(* IEC 61131-3 sources: traffic-lights/PLC_TrafficLights/Class/SdiasManager (part 4) *)

    if pAccessHandle then
      pAccessHandle^ := 0;
    end_if;

    Success := FALSE;
  end_if;

END_FUNCTION

FUNCTION VIRTUAL SdiasManager::AddBroadCastAccessesToList
  VAR
    i : USINT;
  END_VAR

  // Memory for Access data is already held by SDIAS Manager, No need for pHelpAccess

  // count the data for the varan payload frames
  // Access type is control broadcast 2 Byte, Read 0 Byte
  if SupportedFeatures.TimeBroadCastSupported then
    for i := 0 to SDIAS_NR_TIMEBROADCAST_DOS - 1 do
      ISOWriteDO.Length += sizeof(t_SDIAS_ControlByte) + sizeof(UINT);  // control byte + data length
      ISOReadDO.Length  += sizeof(t_SDIAS_StateByte);                   // state byte
    end_for;
  end_if;

END_FUNCTION

FUNCTION VIRTUAL SdiasManager::CheckTimeBroadCastSupported
	VAR_OUTPUT
		bTimeBroadCastSupported 	: BOOL;
	END_VAR
  VAR
    tempCmd             : CmdStruct;
    _result             : results;
    retval              : iprStates;
  END_VAR

  // Countercheck
  bTimeBroadCastSupported := TRUE;

  // Check if broadcast command is supported by OS
  if ConnectionType = SDIAS_CON_LOCAL_uC then

    // OS is only needed for local SDIAS
    if (pSDIAS^.udVersion < SDIAS_CILVERSION_BROADCAST) then
      bTimeBroadCastSupported := FALSE;
    end_if;

  end_if;

  // Check if broadcast command is supported SDIAS Manager
  if FeatureInfo.ProtocolVersion < SDIAS_PROTOCOLVERSION_BROADCAST then
    bTimeBroadCastSupported := FALSE;
  end_if;

  // Timestamp of HWControl must be valid
  tempCmd.uiCmd := CMD_GET_HW_TIMESTAMP;
  tempCmd.aPara[0]$t_GetHwTimestampCmd.udVersion    := 1;
  tempCmd.aPara[0]$t_GetHwTimestampCmd.udCoreSelect := 0;

  _result.aData[0]$t_GetHwTimestampResult.udVersion := 0; // Init return Value incase command is not implemented in HWControl

  retval := ToBusInterface.NewInst(#tempCmd, #_result);

  if retval <> READY then
    bTimeBroadCastSupported := FALSE;
  elsif _result.aData[0]$t_GetHwTimestampResult.udVersion < 1 then
    bTimeBroadCastSupported := FALSE;
  end_if;

END_FUNCTION

FUNCTION VIRTUAL SdiasManager::ReceiveSDOResponse
	VAR_INPUT
		Command 	: t_SDIAS_SDO_Cmd;
		Offset 	: HINT;
		Length 	: USINT;
		Result 	: iprStates;
		pResponseBuffer 	: ^USINT;
		ResponseLength 	: USINT;
	END_VAR
	VAR_OUTPUT
		ret_code 	: iprStates;
	END_VAR

  ret_code := READY;

  case Command of
    SDIAS_SDO_CMD_REBUILD_SDIAS:
      // if it succeeded, check if we have something to do
      if Result = READY then
        // everthing is fine
      else
        // an error occured while performing the operation
#ifdef HWC_LogError
        HWC_LogError(this, "@0083 (SdiasManager::ReceiveSDOResponse) Rebuild SDIAS SDO command failed!");
#endif
      end_if;
    SDIAS_SDO_CMD_SET_NEW_END:
      // if it succeeded, check if we have something to do
      if Result = READY then
        // everthing is fine
        bReceivedNewEndRsp := TRUE;
      else
        // an error occured while performing the operation
#ifdef HWC_LogError
        HWC_LogError(this, "@0084 (SdiasManager::ReceiveSDOResponse) Set new DOL end command failed!");
#endif
      end_if;

  else
    ret_code := ERROR;
#ifdef HWC_LogError
    HWC_LogError(this, "@0085 (SdiasManager::ReceiveSDOResponse) Invalid command in SDO response!");
#endif
  end_case;

END_FUNCTION

FUNCTION VIRTUAL SdiasManager::AddSDOReq
	VAR_INPUT
		pCmdSvr 	: ^SvrChCmd;
		Command 	: t_SDIAS_SDO_Cmd;
		Place 	: USINT;
		CmdLength 	: USINT;
		pReqBuf 	: ^USINT;
	END_VAR
	VAR_OUTPUT
		sd_retval 	: DINT;
	END_VAR

  // protect via mutex because this can be called from different task priorities
  OS_MT_WAIT(pv_Mutex);

  // if the buffer is full, or the next element in the buffer is already in use
  if (SDOHandling.pWrite^.Command <> SDIAS_SDO_CMD_INVALID) then
    sd_retval := SDIAS_MAILBOX_FULL;
    OS_MT_SIGNAL(pv_Mutex);
    return;
  end_if;

  // check the pointer first (if needed)
  if CmdLength then
    if pReqBuf then
      _memcpy(ptr1:=#SDOHandling.pWrite^.ReqBufData, ptr2:=pReqBuf, cntr:=CmdLength);
    else
      sd_retval := SDIAS_INVALID_PARAM_DATA_BUFFER;
      OS_MT_SIGNAL(pv_Mutex);
      return;
    end_if;
  end_if;

  SDOHandling.pWrite^.pCallBackSvr := pCmdSvr;
  SDOHandling.pWrite^.NMTCommand := 0;
  SDOHandling.pWrite^.SDIASPlace := Place;
  SDOHandling.pWrite^.CmdLength := CmdLength;

  case Command of
    SDIAS_SDO_CMD_MEM_READ,
    SDIAS_SDO_CMD_MEM_WRITE,
    SDIAS_SDO_CMD_CTRL_READ,
    SDIAS_SDO_CMD_CTRL_WRITE:
//    SDIAS_SDO_CMD_SPI_READ,
//    SDIAS_SDO_CMD_SPI_WRITE:
      // store offset and length for read and write accesses
      SDOHandling.pWrite^.RdWrHead := pReqBuf^$t_SDIAS_SDO_RdWr_Head;
    SDIAS_SDO_CMD_SPI_READ,
    SDIAS_SDO_CMD_SPI_WRITE:

      // store offset and length for read and write accesses
      SDOHandling.pWrite^.RdWrHead := pReqBuf^$t_SDIAS_SDO_RdWr_Head;

  end_case;

  // command is the last thing to store, because it indicates a complete entry
  SDOHandling.pWrite^.Command := Command;

  // we increment our used entries in the buffer (only for debugging)
  SDOHandling.EntriesUsed     += 1;

  // after we successfully added this SDO, set the write pointer to the next element
  if SDOHandling.pWrite = SDOHandling.pLastEntry then
    SDOHandling.pWrite := SDOHandling.pRingBufMemStart;
  else
    SDOHandling.pWrite += sizeof(t_SDORingBufEntry);
  end_if;

  sd_retval := SDIAS_OK;

  OS_MT_SIGNAL(pv_Mutex);

END_FUNCTION

FUNCTION VIRTUAL SdiasManager::CyclicSDOHandling
  VAR
  	i,j           : USINT;
    FoundIt       : BOOL;
		Offset 	      : HINT;
		Length 	      : USINT;
    pTempChannel  : ^t_SDOChannel;
    TempChannel   : t_SDOChannel;
    pRingBufEntry : ^t_SDORingBufEntry;
    FirstFound    : USINT;
    LastFound     : USINT;
    Channels2Add  : DINT;
    StartIndex    : USINT;
    EndIndex      : USINT;
    pCmdSvr       : ^SvrChCmd;
  	tempCmd       : CmdStruct;
    _result       : results;
    ReceiveBuffer : ARRAY [0..127] OF USINT;
    ReceiveLength : UDINT;
    sd_retval     : DINT;
    TempUDINT     : UDINT;
    OldChannelNo  : USINT;
  END_VAR

  // protect via mutex because this can be called from different task priorities
  OS_MT_WAIT(pv_Mutex);

  if ConnectionType = SDIAS_CON_VIA_VARAN_uC then

    // check sdo response first. if a channel is ready it can be used for the next request

    // GET SDO RESPONSE
    if (AsyReadUsage = _NotUsed) | (AsyReadUsage = _UsedBySDO) then

      // if the AsyRdDO is used for polling, we check if we got a response
      if AsyReadUsage = _UsedBySDO then
        StartIndex := ((ASYReadDO.Offset - SDOHandling.OffsetSDOResp) / sizeof(t_SDOChannel))$USINT;
        EndIndex := StartIndex + (ASYReadDO.Length / sizeof(t_SDOChannel))$USINT - 1;
        Offset := 0;
        for i := StartIndex to EndIndex do
          if SDOHandling.aChannelData[i].WaitForResponse then
            // check for the response (copy only header first)
            _memcpy(ptr1:=#TempChannel, ptr2:=ASYReadDO.pData$^t_SDOChannel + Offset, cntr:=sizeof(t_SDOChannel) - sizeof(t_SDOChannel.Data));
            pRingBufEntry := SDOHandling.aChannelData[i].pActElement;

            // if the header info is mirrored, the SDO is ready
            if ((TempChannel.MessageCounter AND SDIAS_MASK_MESSAGE_COUNTER) = pRingBufEntry^.MessageCounter) &
               (TempChannel.SDIASPlace = pRingBufEntry^.SDIASPlace) &
               (TempChannel.Command$t_SDIAS_SDO_Cmd = pRingBufEntry^.Command) then

              // we got our response
              SDOHandling.aChannelData[i].WaitForResponse := FALSE;
              SDOHandling.EntriesUsed -= 1;

              // check for error
              if (TempChannel.MessageCounter AND SDIAS_MASK_GLOBAL_ERROR_FLAG) then
                tempCmd.aPara[3] := ERROR;
                // copy error info
                _memcpy(ptr1:=#TempChannel.Data, ptr2:=ASYReadDO.pData + t_SDOChannel.Data + Offset, cntr:=TempChannel.LengthOfData);

                // show error info
                case TempChannel.Data$DINT of
                  SDIAS_SDO_ERROR_INVALID_MSG_CNT:
#ifdef HWC_LogValue1
                    HWC_LogValue1(this, "@0086 (SdiasManager::CyclicSDOHandling) SDO Error 0x{0}: Invalid message counter", TempChannel.Data$UDINT);
#endif

                  SDIAS_SDO_ERROR_MSG_CNT_NOT_SUCCESSIVE:
#ifdef HWC_LogValue1
                    HWC_LogValue1(this, "@0087 (SdiasManager::CyclicSDOHandling) SDO Error 0x{0}: Message counter not successive", TempChannel.Data$UDINT);
#endif

                  SDIAS_SDO_ERROR_INVALID_CMD:
#ifdef HWC_LogValue1
                    HWC_LogValue1(this, "@0088 (SdiasManager::CyclicSDOHandling) SDO Error 0x{0}: Invalid command", TempChannel.Data$UDINT);
#endif

                  SDIAS_SDO_ERROR_INVALID_SUBCMD:
#ifdef HWC_LogValue1
                    HWC_LogValue1(this, "@0089 (SdiasManager::CyclicSDOHandling) SDO Error 0x{0}: Invalid subcommand", TempChannel.Data$UDINT);
#endif

                  SDIAS_SDO_ERROR_INVALID_PLACE:
#ifdef HWC_LogValue1
                    HWC_LogValue1(this, "@008A (SdiasManager::CyclicSDOHandling) SDO Error 0x{0}: Invalid SDIAS Place", TempChannel.Data$UDINT);
#endif

                  SDIAS_SDO_ERROR_INVALID_CMD_LENGTH:
#ifdef HWC_LogValue1
                    HWC_LogValue1(this, "@008B (SdiasManager::CyclicSDOHandling) SDO Error 0x{0}: Invalid length of data bytes", TempChannel.Data$UDINT);
#endif

                  SDIAS_SDO_ERROR_INVALID_ACCESS_OFFSET:
#ifdef HWC_LogValue1
                    HWC_LogValue1(this, "@008C (SdiasManager::CyclicSDOHandling) SDO Error 0x{0}: Invalid offset for access", TempChannel.Data$UDINT);
#endif

                  SDIAS_SDO_ERROR_INVALID_ACCESS_LENGTH:
#ifdef HWC_LogValue1
                    HWC_LogValue1(this, "@008D (SdiasManager::CyclicSDOHandling) SDO Error 0x{0}: Invalid length for access", TempChannel.Data$UDINT);
#endif

                  SDIAS_SDO_ERROR_INTERNAL_TIMEOUT:
#ifdef HWC_LogValue1
                    HWC_LogValue1(this, "@008E (SdiasManager::CyclicSDOHandling) SDO Error 0x{0}: Internal timeout", TempChannel.Data$UDINT);
#endif

                  SDIAS_SDO_ERROR_GENERAL_ERROR:
#ifdef HWC_LogValue1
                    HWC_LogValue1(this, "@008F (SdiasManager::CyclicSDOHandling) SDO Error 0x{0}: General Error", TempChannel.Data$UDINT);
#endif

                  SDIAS_SDO_ERROR_MSG_CNT_CHANGED:
#ifdef HWC_LogValue1
                    HWC_LogValue1(this, "@0090 (SdiasManager::CyclicSDOHandling) SDO Error 0x{0}: Message counter changed while SDO request was processed", TempChannel.Data$UDINT);
#endif

                  SDIAS_SDO_ERROR_CLIENT_NOT_READY:
#ifdef HWC_LogValue1
                    HWC_LogValue1(this, "@0091 (SdiasManager::CyclicSDOHandling) SDO Error 0x{0}: Communication error between SDIAS Manager and SDIAS Client", TempChannel.Data$UDINT);
#endif

                  SDIAS_SDO_ERROR_MNG_DPRAM_FAILURE:
#ifdef HWC_LogValue1
                    HWC_LogValue1(this, "@0092 (SdiasManager::CyclicSDOHandling) SDO Error 0x{0}: Error accessing the SDIAS Manager DPRAM", TempChannel.Data$UDINT);
#endif

                  SDIAS_SDO_ERROR_ACCESS_NOT_ALLOWED:
#ifdef HWC_LogValue1
                    HWC_LogValue1(this, "@0093 (SdiasManager::CyclicSDOHandling) SDO Error 0x{0}: Access not allowed (e.g. control access to SDIAS Manager)", TempChannel.Data$UDINT);
#endif

                  SDIAS_SDO_ERROR_FLASH_ACCESS_FAILED:
#ifdef HWC_LogValue1
                    HWC_LogValue1(this, "@0094 (SdiasManager::CyclicSDOHandling) SDO Error 0x{0}: Flash access failed", TempChannel.Data$UDINT);
#endif

                  SDIAS_SDO_ERROR_INVALID_PARAMETERS:
#ifdef HWC_LogValue1
                    HWC_LogValue1(this, "@0095 (SdiasManager::CyclicSDOHandling) SDO Error 0x{0}: Invalid parameters in SDO request", TempChannel.Data$UDINT);
#endif

                else
#ifdef HWC_LogValue1
                  HWC_LogValue1(this, "@0096 (SdiasManager::CyclicSDOHandling) SDO Error 0x{0}: Unknown Error", TempChannel.Data$UDINT);
#endif
                end_case;
              else
                tempCmd.aPara[3]$iprStates := READY;
                // copy response data
                if TempChannel.LengthOfData then
                  if TempChannel.LengthOfData <= sizeof(t_SDOChannel.Data) then
                    _memcpy(ptr1:=#TempChannel.Data, ptr2:=ASYReadDO.pData + t_SDOChannel.Data + Offset, cntr:=TempChannel.LengthOfData);
                  else
#ifdef HWC_LogValue2
                    HWC_LogValue2(this, "@0097 (SdiasManager::CyclicSDOHandling) SDO Error: Length in response is too big (0x{0} Byte; Max: 0x{1} Byte)", TempChannel.LengthOfData, sizeof(t_SDOChannel.Data));
#endif
                  end_if;
                end_if;
              end_if;

              // if there is a response, distribute it and set this channel to "available for the next SDO" (set command to SDIAS_SDO_CMD_INVALID and pChannel to NIL)
              tempCmd.uiCmd := SDIAS_CMD_SDO_RESPONSE;
              tempCmd.aPara[0] := TempChannel.Command$t_SDIAS_SDO_Cmd;

              // if we got response data
              if TempChannel.LengthOfData then

                // if the SDO command was successful
                if tempCmd.aPara[3]$iprStates = READY then

                  // check if it's a command with offset and length info
                  case TempChannel.Command$t_SDIAS_SDO_Cmd of
                    SDIAS_SDO_CMD_MEM_READ,
                    SDIAS_SDO_CMD_MEM_WRITE,
                    SDIAS_SDO_CMD_CTRL_READ,
                    SDIAS_SDO_CMD_CTRL_WRITE:
                      // save header info in extra parameters
                      tempCmd.aPara[1] := pRingBufEntry^.RdWrHead.Offset;
                      tempCmd.aPara[2] := pRingBufEntry^.RdWrHead.Length;

                      // remove header info for user from payload
                      TempChannel.LengthOfData -= sizeof(t_SDIAS_SDO_RdWr_Head);

                      // pointer to data
                      tempCmd.aPara[4] := (#TempChannel.Data + sizeof(t_SDIAS_SDO_RdWr_Head))$DINT;

                    SDIAS_SDO_CMD_SPI_READ,
                    SDIAS_SDO_CMD_SPI_WRITE:

                      // no length or offset available
                      tempCmd.aPara[1] := 0;
                      tempCmd.aPara[2] := 0;

                      // pointer to data
                      tempCmd.aPara[4] := (#TempChannel.Data)$DINT;

                  else
                      // no length or offset available
                      tempCmd.aPara[1] := 0;
                      tempCmd.aPara[2] := 0;

                      // pointer to data
                      tempCmd.aPara[4] := (#TempChannel.Data)$DINT;
                  end_case;
                else
                  // check if it's a command with offset and length info
                  case TempChannel.Command$t_SDIAS_SDO_Cmd of
                    SDIAS_SDO_CMD_MEM_READ,
                    SDIAS_SDO_CMD_MEM_WRITE,
                    SDIAS_SDO_CMD_CTRL_READ,
                    SDIAS_SDO_CMD_CTRL_WRITE,
                    SDIAS_SDO_CMD_SPI_READ,
                    SDIAS_SDO_CMD_SPI_WRITE:
                      // save header info in extra parameters
                      tempCmd.aPara[1] := pRingBufEntry^.RdWrHead.Offset;
                      tempCmd.aPara[2] := pRingBufEntry^.RdWrHead.Length;
                  end_case;

                  // pointer to error code
                  tempCmd.aPara[4] := (#TempChannel.Data)$DINT;
                end_if;
              else
                tempCmd.aPara[4] := 0;
              end_if;
              tempCmd.aPara[5] := TempChannel.LengthOfData;

              pCmdSvr := pRingBufEntry^.pCallBackSvr;

              if pCmdSvr$pVirtualBase^.NewInst(#tempCmd, #_result) <> READY then
#ifdef HWC_LogValue1
                HWC_LogValue1(this, "@0099 (SdiasManager::CyclicSDOHandling) SDO Error: Error of module at place 0x{0} while receiving the SDO reponse (which was an ErrorCode)", i);
#endif
              end_if;

              // the position in the ringbuffer is free again
              pRingBufEntry^.BusyChannelNo := 0;
              pRingBufEntry^.Command := SDIAS_SDO_CMD_INVALID;

              // the SDO channel on the module is free again
              SDOHandling.aChannelData[i].pActElement := NIL;

            elsif (ops.tAbsolute - SDOHandling.aChannelData[i].RequestTime) >= SDIAS_SDO_TIMEOUT then
              // the SDO request timed out (should not happen)
#ifdef HWC_LogValue1
              HWC_LogValue1(this, "@0098 (SdiasManager::CyclicSDOHandling) SDO Error: Timeout while waiting for answer of the SDIAS Manager µC (Channel {0} of range 1-3)", i+1);
#endif

              // we got our response
              SDOHandling.aChannelData[i].WaitForResponse := FALSE;
              SDOHandling.EntriesUsed -= 1;

              // distribute timeout error and set this channel to "available for the next SDO" (set command to SDIAS_SDO_CMD_INVALID and pChannel to NIL)
              tempCmd.uiCmd := SDIAS_CMD_SDO_RESPONSE;
              tempCmd.aPara[0] := pRingBufEntry^.Command$UINT;

              // check if it's a command with offset and length info
              case pRingBufEntry^.Command of
                SDIAS_SDO_CMD_MEM_READ,
                SDIAS_SDO_CMD_MEM_WRITE,
                SDIAS_SDO_CMD_CTRL_READ,
                SDIAS_SDO_CMD_CTRL_WRITE,
                SDIAS_SDO_CMD_SPI_READ,
                SDIAS_SDO_CMD_SPI_WRITE:
                  // save header info in extra parameters
                  tempCmd.aPara[1] := pRingBufEntry^.RdWrHead.Offset;
                  tempCmd.aPara[2] := pRingBufEntry^.RdWrHead.Length;
              else
                  // no length or offset available
                  tempCmd.aPara[1] := 0;
                  tempCmd.aPara[2] := 0;
              end_case;

              tempCmd.aPara[3] := ERROR;
              tempCmd.aPara[4] := 0;
              tempCmd.aPara[5] := 0; // no data available

              pCmdSvr := pRingBufEntry^.pCallBackSvr;
              if pCmdSvr$pVirtualBase^.NewInst(#tempCmd, #_result) <> READY then
#ifdef HWC_LogValue1
                HWC_LogValue1(this, "@0099 (SdiasManager::CyclicSDOHandling) SDO Error: Error of module at place 0x{0} while receiving the SDO reponse", i);
#endif
              end_if;

              // the position in the ringbuffer is free again
              pRingBufEntry^.BusyChannelNo := 0;
              pRingBufEntry^.Command := SDIAS_SDO_CMD_INVALID;

              // the SDO channel on the module is free again
              SDOHandling.aChannelData[i].pActElement := NIL;
            end_if;
          end_if;

          Offset += sizeof(t_SDOChannel);
        end_for;
      end_if;

      // check for the first (needed for offset) and last (needed for length)
      Length := 0;
      FoundIt := FALSE;
      for i := 0 to (SDIAS_SDO_CHANNEL_NO-1) do
        if SDOHandling.aChannelData[i].pActElement & SDOHandling.aChannelData[i].WaitForResponse then
          if FoundIt = FALSE then
            // found first used channel
            FoundIt := TRUE;
            Offset := SDOHandling.OffsetSDOResp + i * sizeof(t_SDOChannel);
          end_if;
          Length += sizeof(t_SDOChannel);
        end_if;
      end_for;

      if FoundIt then

        // if we have pending SDO requests, start the AsyRdDO for polling
        if ChangeAsyRd(Offset:=Offset,
                       Length:=Length,
                       RunState:=_BUS_IF_RUN_STATE_CONT_RUN,
                       UsageType:=_UsedBySDO) = FALSE then
#ifdef HWC_LogError
          HWC_LogError(this, "@009A (SdiasManager::CyclicSDOHandling) Error occured at starting the ReadDO for SDO polling");
#endif
        end_if;
      else
        // if all pending SDOs received stop DO
        if AsyReadUsage = _UsedBySDO then
          if ChangeAsyRd(Offset:=0,
                         Length:=0,
                         RunState:=_BUS_IF_RUN_STATE_NO_RUN,
                         UsageType:=_UsedBySDO) = FALSE then
#ifdef HWC_LogError
          HWC_LogError(this, "@009B (SdiasManager::CyclicSDOHandling) Error occured at stopping the ReadDO");
#endif
          end_if;
        end_if;
      end_if;
    end_if;

    // SEND SDO REQUEST
    if (AsyWriteUsage = _NotUsed) | (AsyWriteUsage = _UsedBySDO) then
      // if there is a free channel on the module, we have unsent requests and the AsyWrDO is not used => send the Request (or more than 1 if possible)

      // first check if we need to increment the msg counter for a previously sent SDO message
      if SDOHandling.IncrementMsgCnt then
        for i := 0 to (SDIAS_SDO_CHANNEL_NO-1) do
          if SDOHandling.IncrementMsgCnt AND 1 then
            // next message counter for this channel
            if SDOHandling.aChannelData[i].MessageCnt = SDIAS_MASK_MESSAGE_COUNTER then
              SDOHandling.aChannelData[i].MessageCnt    := 0;
            else
              SDOHandling.aChannelData[i].MessageCnt    += 1;
            end_if;

            SDOHandling.aChannelData[i].pActElement^.MessageCounter := SDOHandling.aChannelData[i].MessageCnt;
            pTempChannel := #SDOHandling.aChannelData[i].ChannelData;
            pTempChannel^.MessageCounter  := SDOHandling.aChannelData[i].MessageCnt;

            // save the new message counter to the Varan DO
            _memcpy(ptr1:=ASYWriteDO.pData$^USINT + i * sizeof(t_SDOChannel) - (ASYWriteDO.Offset - SDOHandling.OffsetSDOReq)$USINT, ptr2:=pTempChannel, cntr:=pTempChannel^.LengthOfData + sizeof(t_SDOChannel) - sizeof(t_SDOChannel.Data));
            SDOHandling.aChannelData[i].WaitForResponse := TRUE;
            TempUDINT := ops.tAbsolute;
            SDOHandling.aChannelData[i].RequestTime     := TempUDINT;
          end_if;
          SDOHandling.IncrementMsgCnt := SDOHandling.IncrementMsgCnt SHR 1;
        end_for;

        // use the same length and offset (it's the same frame just with different message counters)
        Offset := ASYWriteDO.Offset;
        Length := ASYWriteDO.Length$USINT;

        // write the same frame again with higher message counter on the modified SDOs
        if ChangeAsyWr(Offset:=Offset,
                       Length:=Length,
                       RunState:=_BUS_IF_RUN_STATE_CONT_RUN,
                       UsageType:=_UsedBySDO) = FALSE then
#ifdef HWC_LogError
          HWC_LogError(this, "@009C (SdiasManager::CyclicSDOHandling) Error occured at starting the WriteDO to write the new message counter");
#endif
        end_if;
      else
        // check for a free channel
        FoundIt := FALSE;
        for i := 0 to (SDIAS_SDO_CHANNEL_NO-1) do
          if SDOHandling.aChannelData[i].pActElement = NIL then
            // found a free channel
            FoundIt := TRUE;
            FirstFound := LastFound := i;
            Offset := SDOHandling.OffsetSDOReq + i * sizeof(t_SDOChannel);
            exit;
          end_if;
        end_for;

        // now we fill the buffer in the channels of the hardware (continue as long as there is space in the buffer and we have SDOs to send)
        Channels2Add := 0;
        while FoundIt & (SDOHandling.pRead^.Command <> SDIAS_SDO_CMD_INVALID) & (SDOHandling.pRead^.BusyChannelNo = 0) do
          // i is the index of the free channel => add the data
          pTempChannel := #SDOHandling.aChannelData[i].ChannelData;
          SDOHandling.aChannelData[i].pActElement     := SDOHandling.pRead;
          SDOHandling.pRead^.MessageCounter           := SDOHandling.aChannelData[i].MessageCnt;
          pTempChannel^.MessageCounter                := SDOHandling.pRead^.MessageCounter;
          pTempChannel^.NMT                           := SDOHandling.pRead^.NMTCommand;
          pTempChannel^.SDIASPlace                    := SDOHandling.pRead^.SDIASPlace;
          pTempChannel^.Command$t_SDIAS_SDO_Cmd       := SDOHandling.pRead^.Command;
          pTempChannel^.LengthOfData                  := SDOHandling.pRead^.CmdLength;
          if pTempChannel^.LengthOfData then
            _memcpy(ptr1:=#pTempChannel^.Data, ptr2:=#SDOHandling.pRead^.ReqBufData, cntr:=pTempChannel^.LengthOfData);
          end_if;

          // put the SDO request into the DPRAM on the right channel
          _memcpy(ptr1:=ASYWriteDO.pData$^t_SDOChannel + Channels2Add * sizeof(t_SDOChannel), ptr2:=pTempChannel, cntr:=pTempChannel^.LengthOfData + sizeof(t_SDOChannel) - sizeof(t_SDOChannel.Data));

          // remember this as the last found SDO to work with
          LastFound := i;

          // remember that we have to increment the message counter here
          SDOHandling.IncrementMsgCnt := SDOHandling.IncrementMsgCnt OR (1 SHL i);

          // this element is done by channel x
          SDOHandling.pRead^.BusyChannelNo := i+1;

          // increase channels to add
          Channels2Add += 1;

          // after we successfully added this SDO, set the read pointer to the next element
          if SDOHandling.pRead = SDOHandling.pLastEntry then
            SDOHandling.pRead := SDOHandling.pRingBufMemStart;
          else
            SDOHandling.pRead += sizeof(t_SDORingBufEntry);
          end_if;

          OldChannelNo := i;

          // check for a free channel
          FoundIt := FALSE;
          for i := 0 to (SDIAS_SDO_CHANNEL_NO-1) do
            if SDOHandling.aChannelData[i].pActElement = NIL then
              // found a free channel
              FoundIt := TRUE;

              if i > (OldChannelNo + 1) then
                // refresh the data in the DPRAM for the skipped channels
                for j := (OldChannelNo+1) to (i-1) do
                  // put the SDO request into the DPRAM on the right channel
                  _memcpy(ptr1:=ASYWriteDO.pData$^t_SDOChannel + j * sizeof(t_SDOChannel), ptr2:=#SDOHandling.aChannelData[j].ChannelData, cntr:=SDOHandling.aChannelData[j].ChannelData.LengthOfData + sizeof(t_SDOChannel) - sizeof(t_SDOChannel.Data));

                  // increase channels to add, because we also write the skipped ones
                  Channels2Add += 1;
                end_for;
              end_if;

              exit;
            end_if;
          end_for;
        end_while;

        if Channels2Add then
          Length := (LastFound - FirstFound + 1)$USINT * sizeof(t_SDOChannel);
          // if we have something to write => write it
          if ChangeAsyWr(Offset:=Offset,
                         Length:=Length,
                         RunState:=_BUS_IF_RUN_STATE_CONT_RUN,
                         UsageType:=_UsedBySDO) = FALSE then
#ifdef HWC_LogError
            HWC_LogError(this, "@009D (SdiasManager::CyclicSDOHandling) Error occured at starting the WriteDO to write the new SDO command");
#endif
          end_if;
        elsif AsyWriteUsage = _UsedBySDO then
          // otherwise release the write buffer to other purposes
          if ChangeAsyWr(Offset:=0,
                         Length:=0,
                         RunState:=_BUS_IF_RUN_STATE_NO_RUN,
                         UsageType:=_UsedBySDO) = FALSE then
#ifdef HWC_LogError
            HWC_LogError(this, "@009E (SdiasManager::CyclicSDOHandling) Error occured at stopping the WriteDO");
#endif
          end_if;
        end_if;
      end_if;
    end_if;
  else
    // if connected locally we can use the OS interfaces to access the SDO channels

    // check sdo response first. if a channel is ready it can be used for the next request

    // GET SDO RESPONSE
    if SDOHandling.EntriesUsed then
      // post init blocks the tasks in cyclic priority (the SDIAS Manager Code is running in lower priority than cyclic and has no time during the postinit) => give it some time
      if (b_PostInitFinished = FALSE) then
        ToMultiTask.TASKDELAY(timeout0:=SDIAS_WAIT_TIME_IN_POST_INIT);
      end_if;
      // check if we got a response
      for i := 0 to (SDIAS_SDO_CHANNEL_NO-1) do
        if SDOHandling.aChannelData[i].WaitForResponse then

          // get the SDO response
          ReceiveLength := 0;
          sd_retval := SDIAS_iReadSdoResponseChannel(udSdoHandle       := SDOHandling.aChannelData[i].SdoHandle
                                                   , udBufferLength    := sizeof(ReceiveBuffer)
                                                   , pucData           := #ReceiveBuffer[0]
                                                   , pudDataLength     := #ReceiveLength
                                                   );

          // check if it's finished => no more busy
          if sd_retval <> SDIAS_SDO_REQUEST_BUSY then
            if ReceiveLength <= sizeof(TempChannel.Data) then
              pRingBufEntry := SDOHandling.aChannelData[i].pActElement;

              // copy the info
              _memcpy(ptr1:= #TempChannel.Data, ptr2:= #ReceiveBuffer[0], cntr:= ReceiveLength);
              TempChannel.LengthOfData := ReceiveLength$USINT;
              TempChannel.Command$t_SDIAS_SDO_Cmd := pRingBufEntry^.Command;

              // we got our response
              SDOHandling.aChannelData[i].WaitForResponse := FALSE;
              SDOHandling.EntriesUsed -= 1;

              // check for error
              if sd_retval <> SDIAS_OK then
                tempCmd.aPara[3] := ERROR;

                LogSDOErrorInfo(sd_retval);
              else
                tempCmd.aPara[3]$iprStates := READY;
              end_if;

              // if there is a response, distribute it and set this channel to "available for the next SDO" (set command to SDIAS_SDO_CMD_INVALID and pChannel to NIL)
              tempCmd.uiCmd := SDIAS_CMD_SDO_RESPONSE;
              tempCmd.aPara[0] := pRingBufEntry^.Command$INT;

              // if we got response data
              if TempChannel.LengthOfData then

                // if the SDO command was successful
                if tempCmd.aPara[3]$iprStates = READY then

                  // check if it's a command with offset and length info
                  case TempChannel.Command$t_SDIAS_SDO_Cmd of
                    SDIAS_SDO_CMD_MEM_READ,
                    SDIAS_SDO_CMD_MEM_WRITE,
                    SDIAS_SDO_CMD_CTRL_READ,
                    SDIAS_SDO_CMD_CTRL_WRITE:
                      // save header info in extra parameters
                      tempCmd.aPara[1] := pRingBufEntry^.RdWrHead.Offset;
                      tempCmd.aPara[2] := pRingBufEntry^.RdWrHead.Length;

                      // remove header info for user from payload
                      TempChannel.LengthOfData -= sizeof(t_SDIAS_SDO_RdWr_Head);

                      // pointer to data
                      tempCmd.aPara[4] := (#TempChannel.Data + sizeof(t_SDIAS_SDO_RdWr_Head))$DINT;

                    SDIAS_SDO_CMD_SPI_READ,
                    SDIAS_SDO_CMD_SPI_WRITE:
                      // no length or offset available
                      tempCmd.aPara[1] := 0;
                      tempCmd.aPara[2] := 0;

                      // pointer to data
                      tempCmd.aPara[4] := (#TempChannel.Data)$DINT;

                  else
                      // no length or offset available
                      tempCmd.aPara[1] := 0;
                      tempCmd.aPara[2] := 0;

                      // pointer to data
                      tempCmd.aPara[4] := (#TempChannel.Data)$DINT;
                  end_case;
                else
                  // check if it's a command with offset and length info
                  case TempChannel.Command$t_SDIAS_SDO_Cmd of
                    SDIAS_SDO_CMD_MEM_READ,
                    SDIAS_SDO_CMD_MEM_WRITE,
                    SDIAS_SDO_CMD_CTRL_READ,
                    SDIAS_SDO_CMD_CTRL_WRITE,
                    SDIAS_SDO_CMD_SPI_READ,
                    SDIAS_SDO_CMD_SPI_WRITE:
                      // save header info in extra parameters
                      tempCmd.aPara[1] := pRingBufEntry^.RdWrHead.Offset;
                      tempCmd.aPara[2] := pRingBufEntry^.RdWrHead.Length;
                  end_case;

                  // pointer to error code
                  tempCmd.aPara[4] := (#sd_retval)$DINT;
                end_if;
              else
                tempCmd.aPara[4] := 0;
              end_if;
              tempCmd.aPara[5] := TempChannel.LengthOfData;

              pCmdSvr := pRingBufEntry^.pCallBackSvr;
              if pCmdSvr$pVirtualBase^.NewInst(#tempCmd, #_result) <> READY then
#ifdef HWC_LogValue1
                HWC_LogValue1(this, "@0099 (SdiasManager::CyclicSDOHandling) SDO Error: Error of module at place 0x{0} while receiving the SDO reponse (which was an ErrorCode)", i);
#endif
              end_if;

              // the position in the ringbuffer is free again
              pRingBufEntry^.BusyChannelNo := 0;
              pRingBufEntry^.Command := SDIAS_SDO_CMD_INVALID;

              // the SDO channel on the module is free again
              SDOHandling.aChannelData[i].pActElement := NIL;
            else
#ifdef HWC_LogValue2
              HWC_LogValue2(this, "@009F (SdiasManager::CyclicSDOHandling) SDO Response too big. Received 0x{0} bytes. Maximum is 0x{1} bytes.", ReceiveLength, sizeof(TempChannel.Data));
#endif
            end_if;
          end_if;
        end_if;
      end_for;
    end_if;

    // SEND SDO REQUEST
    if SDOHandling.EntriesUsed then
      // if there is a free channel on the module and we have unsent requests => send the Requests

      // check for a free channel
      FoundIt := FALSE;
      for i := 0 to (SDIAS_SDO_CHANNEL_NO-1) do
        if SDOHandling.aChannelData[i].pActElement = NIL then
          // found a free channel
          FoundIt := TRUE;
          FirstFound := LastFound := i;
          exit;
        end_if;
      end_for;

      // now we fill the buffer in the channels of the hardware (continue as long as there is space in the buffer and we have SDOs to send)
      while FoundIt & (SDOHandling.pRead^.Command <> SDIAS_SDO_CMD_INVALID) & (SDOHandling.pRead^.BusyChannelNo = 0) do
        // i is the index of the free channel => add the data
        SDOHandling.aChannelData[i].pActElement     := SDOHandling.pRead;
        SDOHandling.pRead^.MessageCounter           := SDOHandling.aChannelData[i].MessageCnt;
        TempChannel.MessageCounter                  := SDOHandling.pRead^.MessageCounter;
        TempChannel.NMT                             := SDOHandling.pRead^.NMTCommand;
        TempChannel.SDIASPlace                      := SDOHandling.pRead^.SDIASPlace;
        TempChannel.Command$t_SDIAS_SDO_Cmd         := SDOHandling.pRead^.Command;
        TempChannel.LengthOfData                    := SDOHandling.pRead^.CmdLength;
        if TempChannel.LengthOfData then
          _memcpy(ptr1:=#TempChannel.Data, ptr2:=#SDOHandling.pRead^.ReqBufData, cntr:=TempChannel.LengthOfData);
        end_if;

        // send the SDO to the OS Interface
        sd_retval := SDIAS_iSendSdoRequestChannel(hManagerNodeHandle:= udNodeHandle
                                                , udChannel         := i
                                                , udCommand         := TempChannel.Command$t_SDIAS_SDO_Cmd
                                                , udSdiasAddress    := TempChannel.SDIASPlace
                                                , udDataLength      := TempChannel.LengthOfData
                                                , pucData           := #TempChannel.Data[0]
                                                , pudSdoHandle      := #SDOHandling.aChannelData[i].SdoHandle
                                                );

        if sd_retval = SDIAS_OK then
          // this element is done by channel x
          SDOHandling.pRead^.BusyChannelNo := i+1;

          SDOHandling.aChannelData[i].WaitForResponse := TRUE;
          TempUDINT := ops.tAbsolute;
          SDOHandling.aChannelData[i].RequestTime     := TempUDINT;

          // after we successfully added this SDO, set the read pointer to the next element
          if SDOHandling.pRead = SDOHandling.pLastEntry then
            SDOHandling.pRead := SDOHandling.pRingBufMemStart;
          else
            SDOHandling.pRead += sizeof(t_SDORingBufEntry);
          end_if;

          // check for a free channel
          FoundIt := FALSE;
          for i := 0 to (SDIAS_SDO_CHANNEL_NO-1) do
            if SDOHandling.aChannelData[i].pActElement = NIL then
              // found a free channel
              FoundIt := TRUE;
              exit;
            end_if;
          end_for;
        else
          LogSDOErrorInfo(sd_retval);
          exit;
        end_if;
      end_while;
    end_if;
  end_if;

    OS_MT_SIGNAL(pv_Mutex);

END_FUNCTION

FUNCTION VIRTUAL SdiasManager::SetRequiredError
	VAR_INPUT
		pTargetThis 	: ^SdiasBase;(* := NIL *)
		Place 	: UDINT;(* := SDIAS_PLACE_NO_MODULE_ADDED_SO_FAR *)
	END_VAR
  VAR
  	tempCmd         : CmdStruct;
    _result         : results;
    i : UDINT;
    FoundIt : BOOL;
  END_VAR

  if pTargetThis & (Place <> SDIAS_PLACE_NO_MODULE_ADDED_SO_FAR) then
    pTargetThis^.ClassState := _RequiredError;

#ifdef HWC_LogValue1
    HWC_LogValue1(this, "@00A0 (SdiasManager::SetRequiredError) Required Error on SDIAS Place 0x{0}", Place);
#endif
  else
    // general required error (initialisation failed) => search for the first required module to blame (if there is one)
    FoundIt := FALSE;
    if MaxPlace <> SDIAS_PLACE_NO_MODULE_ADDED_SO_FAR then
      for i := 0 to MaxPlace do
        if ModuleObjInfo[i].pThis & ModuleObjInfo[i].Required then
          FoundIt := TRUE;
        end_if;
      end_for;
    end_if;

    // if no required module => don't crash
    if FoundIt = FALSE then
      return;
    end_if;
  end_if;

  ClassState := _RequiredError;

  // set required error
  tempCmd.uiCmd     := _BUS_IF_SET_REQUIRED_ERROR;

  ToBusInterface.NewInst(pPara:=#tempCmd, pResult:=#_result);
  if _result.aData[0]$t_BusIFRetvalErrorcode <> _BUS_IF_RETVAL_OK then
#ifdef HWC_LogError
    HWC_LogError(this, "@00A1 (SdiasManager::SetRequiredError) Failed to set required error to BusInterface");
#endif
  end_if;

  if InitSSW <> _PrepareError then
    ErrorInitStep := InitSSW;
    InitSSW := _PrepareError;
  end_if;

END_FUNCTION

// New interface - 2013-05-28
// -----------------------------------------------------------------------
// -	bIsWriteAcc0 : 0 - read access , 1 - write access
// -	iModAddr0 : Module adress at sdias bus (device adr + offset)
// -	iDataLen0 : Data length
// -	bCtrlAcc0 : 0 - access to regular memory, 1 > access to ctrl access
// -    bAccList0 : 0 - access to iso read/write list, 1 - acc to manager admin list, 2 - access to sdo list, 3 - access to periodic manager list

FUNCTION VIRTUAL SdiasManager::DOL_Handling_Add_DO_TO_List
	VAR_INPUT
		bIsWriteAcc0 	: BOOL;
		usModulePlace0 	: USINT;
		iModAddr0 	: HINT;
		iDataLen0 	: UINT;
		bCtrlAcc0 	: BOOL;
		iWaitDOOffset0 	: UINT;
		bIsDynamic0 	: BOOL;
		pActAccess0 	: ^t_AccessElement;
		bIsBroadCast 	: BOOL;(* := FALSE *)
	END_VAR
	VAR_OUTPUT
		iRetCode 	: DINT;
	END_VAR
  VAR
    pReadList       : ^t_SDIAS_DOL_DESC;
    pWriteList      : ^t_SDIAS_DOL_DESC;
    iEndDataPointRd : UINT;
    iEndDOLPointRd  : UDINT;
    iEndDataPointWr : UINT;
    iEndDOLPointWr  : UDINT;
    udCmdType       : UDINT;
    ReadLen         : UINT;
    ReadAdd         : HDINT;
    WriteLen        : UINT;
    WriteAdd        : HDINT;
    udDOFlags       : UDINT;
    bIsFarAccess    : BOOL;
    usBlockNo1k     : USINT;
    usRetries       : BSINT;
    dolType         : UDINT;
  END_VAR

  iRetCode := -1;

  (* Only ISO DOL	in hardware classes *)
  pReadList := #gcRead_DOL_Desc;
  pWriteList := #gcWrite_DOL_Desc;

  // calculate the module address for far accesses and other
  if pActAccess0^.bIsFarAcc then
    bIsFarAccess  := TRUE;
    usBlockNo1k   := to_usint(iModAddr0 shr 10);
    iModAddr0     := (iModAddr0 AND 16#3FF) + (usModulePlace0 shl 10);
  else
    bIsFarAccess  := FALSE;
    usBlockNo1k   := 0;
    iModAddr0     := iModAddr0 + (usModulePlace0 shl 10);
  end_if;

  if ConnectionType = SDIAS_CON_VIA_VARAN_uC then

    (*	Check endpoints of data and DOL	*)
    iEndDataPointRd := pReadList^.iBaseAddrData + pReadList^.iOffLastData + 1;
    iEndDOLPointRd  := pReadList^.iBaseAddr + pReadList^.iOffEndCmd;

    iEndDataPointWr := pWriteList^.iBaseAddrData + pWriteList^.iOffLastData +  1;
    iEndDOLPointWr  := pWriteList^.iBaseAddr + pWriteList^.iOffEndCmd;

    if(bIsWriteAcc0 = 0) then
      (*	Check endpoints of data and DOL	*)
      iEndDataPointRd += iDataLen0;
      iEndDOLPointRd  += sizeof(t_SDIAS_STD_CMD_DO);
    else
      (*	Check endpoints of data and DOL	*)
      iEndDataPointWr += iDataLen0;
      iEndDOLPointWr  += sizeof(t_SDIAS_STD_CMD_DO);
    end_if;

    (* Check available data	in read space *)
    if(iEndDataPointRd > pReadList^.iEndAddrData) then
      iRetCode := -3;
    (* Check space in DOL	*)
    elsif(iEndDOLPointRd > pReadList^.iEndAddr) then
      iRetCode := -4;
    (* Check available data	in write space *)
    elsif(iEndDataPointWr > pWriteList^.iEndAddrData) then
      iRetCode := -5;
    (* Check space in DOL	*)
    elsif(iEndDOLPointWr > pWriteList^.iEndAddr) then
      iRetCode := -6;
    (* Space for all required data	*)
    else

      // Add 1 to switch to first empty byte
      pWriteList^.iOffLastData += sizeof(t_SDIAS_ControlByte);										(* Add do ctrl byte to data		*)
      pReadList^.iOffLastData += sizeof(t_SDIAS_StateByte);

      pWriteList^.iOffFirstData := pWriteList^.iOffLastData;			(* Store data start points		*)
      pReadList^.iOffFirstData := pReadList^.iOffLastData;

      // dynamic accesses need more bytes in the write payload
      if bIsDynamic0 then
        // control byte is already considered, so we have to add the difference here
        pWriteList^.iOffLastData += (sizeof(t_SDIAS_ControlStructDynamic) - sizeof(t_SDIAS_ControlByte));
      end_if;

      cModulAccessCmds[0].OffsetWritePayload := pWriteList^.iBaseAddrData + pWriteList^.iOffFirstData;		(* Store data offsets			*)
      cModulAccessCmds[0].OffsetReadPayload := pReadList^.iBaseAddrData + pReadList^.iOffFirstData;

      (* Set wait for DO to inactive	*)
      cModulAccessCmds[0].OffsetVolatileWaitFlag := iWaitDOOffset0;

      (* Init scratchpad info to 0	*)
      cModulAccessCmds[0].ErrorInfo := 0;

      usRetries := SDIAS_RETRIES_ALLOWED;
      // No retries with Broadcast
      if bIsBroadCast then
        usRetries := 0;
      end_if;

      (* Ctrl access *)
      if(bCtrlAcc0 <> 0) then
        (* Ctrl access +  retrys	*)
        cModulAccessCmds[0].CmdRetries  := SDIAS_CMD_ACC_CONTROL + (usRetries shl 5);
      elsif bIsFarAccess then
        (* Mem far access +  retrys	*)
        cModulAccessCmds[0].CmdRetries  := SDIAS_CMD_ACC_MEMORY_FAR + (usRetries shl 5);
      else
        (* Mem access +  retrys	*)
        cModulAccessCmds[0].CmdRetries  := SDIAS_CMD_ACC_MEMORY + (usRetries shl 5);
      end_if;

      (* Init reserved info to 0	*)
      cModulAccessCmds[0].Reserved := 0;

      (* Write command to dpram 	*)
      if(bIsWriteAcc0 = 0) then
        if bIsFarAccess then
          cModulAccessCmds[0].ReadLength  := to_usint(iDataLen0);
          cModulAccessCmds[0].ReadOffset  := to_uint(iModAddr0);

          cModulAccessCmds[0].WriteLength := 0;
          cModulAccessCmds[0].WriteOffset := usBlockNo1k;
        else
          cModulAccessCmds[0].ReadLength := to_usint(iDataLen0);
          cModulAccessCmds[0].ReadOffset := to_uint(iModAddr0);

          cModulAccessCmds[0].WriteLength := 0;
          cModulAccessCmds[0].WriteOffset  := 0;
        end_if;

        (* Store write adress of new command  *)
        uiWriteCmdAddr := pReadList^.iBaseAddr + pReadList^.iOffEndCmd;

        (* Increment offset of end command	*)
        pReadList^.iOffEndCmd += sizeof(t_SDIAS_STD_CMD_DO);

        (* End of list	*)
        DOL_Handling_Create_End_Cmd(#cModulAccessCmds[1]);

        (* Add read length to iso read usage	*)
        pReadList^.iOffLastData += iDataLen0;

        (* Set usage vars	*)
        pReadList^.iUsageData := pReadList^.iOffLastData + 1;
        pReadList^.iUsageDOL := pReadList^.iOffEndCmd + sizeof(t_SDIAS_STD_CMD_DO);

        pWriteList^.iUsageData := pWriteList^.iOffLastData + 1;

      else
        if bIsFarAccess then
          cModulAccessCmds[0].ReadLength := 0;
          cModulAccessCmds[0].ReadOffset := usBlockNo1k;

          cModulAccessCmds[0].WriteLength := to_usint(iDataLen0);
          cModulAccessCmds[0].WriteOffset  := to_uint(iModAddr0);
        elsif bIsBroadCast then
          cModulAccessCmds[0]$t_SDIAS_BROADCAST_CMD_DO.iNoOfReadBytes   := 0;
          cModulAccessCmds[0]$t_SDIAS_BROADCAST_CMD_DO.iModAddrRdWrCmd  := to_uint(iModAddr0);
          cModulAccessCmds[0]$t_SDIAS_BROADCAST_CMD_DO.iCmdSubtype      := SDIAS_TIMEBROADCAST_SUBCMD;
          cModulAccessCmds[0]$t_SDIAS_BROADCAST_CMD_DO.iNoOfWriteBytes  := to_usint(iDataLen0);
        else
          cModulAccessCmds[0].ReadLength := 0;
          cModulAccessCmds[0].ReadOffset := 0;

          cModulAccessCmds[0].WriteLength := to_usint(iDataLen0);
          cModulAccessCmds[0].WriteOffset  := to_uint(iModAddr0);
        end_if;

        (* Store write adress of new command  *)
        uiWriteCmdAddr := pWriteList^.iBaseAddr + pWriteList^.iOffEndCmd;

        (* Increment offset of end command	*)
        pWriteList^.iOffEndCmd += sizeof(t_SDIAS_STD_CMD_DO);

        (* End of list	*)
        DOL_Handling_Create_End_Cmd(#cModulAccessCmds[1]);

        (* Add write length to iso write usage	*)
        pWriteList^.iOffLastData += iDataLen0;

        (* Set usage vars	*)
        pReadList^.iUsageData := pReadList^.iOffLastData + 1;

        pWriteList^.iUsageData := pWriteList^.iOffLastData + 1;
        pWriteList^.iUsageDOL := pWriteList^.iOffEndCmd + sizeof(t_SDIAS_STD_CMD_DO);

        (* Reset write payload	*)
        //SDIAS_Module_CPLD_Com_Write_Data(pWriteList^.iBaseAddrData + pWriteList^.iOffFirstData + 1, iDataLen0 , (void *)&iDOL_ResetData[0]);

      end_if;

      iRetCode := 0;

    end_if;

  else
    // locally we use the OS interface to create the DO

    (* Ctrl access *)
    if(bCtrlAcc0 <> 0) then
      (* Ctrl access +  retrys	*)
      udCmdType         := SDIAS_CMD_ACC_CONTROL;
    elsif  bIsFarAccess then
      // far memory access
      udCmdType         := SDIAS_CMD_ACC_MEMORY_FAR;
    else
      (* Mem access +  retrys	*)
      udCmdType         := SDIAS_CMD_ACC_MEMORY;
    end_if;

    // if the interface for dynamic DOs is not available => use the old interface
    if (pSDIAS^.udVersion < SDIAS_CIL_VERSION_SUPPORTS_DYNAMIC_DO) then
      iRetCode := SDIAS_iAddDo(hNodeHandle         := udNodeHandle
                             , udDolType           := SDIAS_DOL_TYPE_ISO
                             , udCmdType           := udCmdType
                             , udRetries           := SDIAS_RETRIES_ALLOWED
                             , udIsWriteAcc        := bIsWriteAcc0
                             , udModuleAddress     := iModAddr0
                             , udDataLen           := iDataLen0
                             , hAddrVolatileWait   := iWaitDOOffset0
                             , phAddrWriteData     := (#cModulAccessCmds[0].OffsetWritePayload)$^pVoid
                             , phAddrReadData      := (#cModulAccessCmds[0].OffsetReadPayload)$^pVoid
                             );

    else

        // make read and write settings
      if bIsWriteAcc0 then
        WriteLen := iDataLen0;
        WriteAdd := iModAddr0;
        ReadLen  := 0;
        ReadAdd  := usBlockNo1k;

        if bIsBroadCast then
          ReadAdd := iModAddr0; // RdWr Access with rd length 0
        end_if;

      else
        WriteLen := 0;
        WriteAdd := usBlockNo1k;
        ReadLen  := iDataLen0;
        ReadAdd  := iModAddr0;
      end_if;

      dolType   := SDIAS_DOL_TYPE_ISO;
      usRetries := SDIAS_RETRIES_ALLOWED;
      // set DO flags
      udDOFlags := 0;
      if bIsDynamic0 then
        if bIsFarAccess then
          udDOFlags := SDIAS_DO_FLAG_SUPPORT_VARIABLE_READ_BYTE_COUNT_AND_MODULE_ADDR OR SDIAS_DO_FLAG_SUPPORT_VARIABLE_WRITE_BYTE_COUNT_AND_MODULE_ADDR;
        else
          if bIsWriteAcc0 then
            udDOFlags := SDIAS_DO_FLAG_SUPPORT_VARIABLE_READ_BYTE_COUNT_AND_MODULE_ADDR;
          else
            udDOFlags := SDIAS_DO_FLAG_SUPPORT_VARIABLE_WRITE_BYTE_COUNT_AND_MODULE_ADDR;
          end_if;
        end_if;
      elsif bIsBroadCast then
        // Set flag for broadcast write to all SDIAS clients
        udDOFlags := SDIAS_DO_FLAG_ACCESS_TYPE_READBROADCASTWRITE_ALL;
        // No retries with Broadcast
        usRetries := 0;
        // Force Broadcast into ISO writelist
        dolType   := SDIAS_DOL_TYPE_ISO_WR;
      end_if;

      // use the new interface
      iRetCode := SDIAS_iAddDoDynamic(hNodeHandle         := udNodeHandle
                                    , udDolType           := dolType
                                    , udCmdType           := udCmdType
                                    , udSubCmdType        := SDIAS_DO_SUBCMD_NONE
                                    , udRetries           := usRetries
                                    , udReadAddress       := ReadAdd
                                    , udReadDataLen       := ReadLen
                                    , udWriteAddress      := WriteAdd
                                    , udWriteDataLen      := WriteLen
                                    , udAddrVolatileWait  := iWaitDOOffset0
                                    , hJumpDoHandle       := SDIAS_INVALID_VOLATILE_WAIT_HANDLE
                                    , udDoFlags           := udDOFlags
                                    , phDoHandle          := #pActAccess0^.udOSDOHandle
                                    , phAddrWriteData     := (#cModulAccessCmds[0].OffsetWritePayload)$^pVoid
                                    , phAddrReadData      := (#cModulAccessCmds[0].OffsetReadPayload)$^pVoid
                                    );
    end_if;

    if iRetCode = SDIAS_OK then
      (* Store data offsets			*)
      pWriteList^.iOffFirstData := cModulAccessCmds[0].OffsetWritePayload - pWriteList^.iBaseAddrData;
      pReadList^.iOffFirstData  := cModulAccessCmds[0].OffsetReadPayload  - pReadList^.iBaseAddrData;
    else
#ifdef HWC_LogError
      HWC_LogError(this, "@00A2 (SdiasManager::DOL_Handling_Add_DO_TO_List) Failed to add custom SDIAS access via OS interface!");
#endif
    end_if;
  end_if;

END_FUNCTION

FUNCTION VIRTUAL SdiasManager::DOL_Handling_Create_End_Cmd
	VAR_INPUT
		pEndCmdBuffer 	: ^t_SDIAS_DOListEntry;
	END_VAR

 	(* End of list	*)
	pEndCmdBuffer^.OffsetReadPayload := 0xFFFF;
	pEndCmdBuffer^.OffsetWritePayload := 0xFFFF;

	(* Set wait for DO to inactive	*)
	pEndCmdBuffer^.OffsetVolatileWaitFlag := SDIAS_INVALID_VOLATILE_WAIT_HANDLE;

	(* Init scratchpad info to 0	*)
	pEndCmdBuffer^.ErrorInfo := 0;

	pEndCmdBuffer^.CmdRetries := 0x0;

	pEndCmdBuffer^.ReadLength := 0;
	pEndCmdBuffer^.ReadOffset := 0;

	(* Init reserved info to 0	*)
	pEndCmdBuffer^.Reserved := 0;

	pEndCmdBuffer^.WriteLength := 0;
	pEndCmdBuffer^.WriteOffset  := 0;

END_FUNCTION

FUNCTION VIRTUAL SdiasManager::LogSDOErrorInfo
	VAR_INPUT
		OSRetVal 	: DINT;
	END_VAR

 // show error info
  case OSRetVal of
    SDIAS_MAILBOX_FULL:
#ifdef HWC_LogValue1
      HWC_LogValue1(this, "@00A3 (SdiasManager::LogSDOErrorInfo) SDO Error 0x{0}: Mailbox full", (0-OSRetVal)$UDINT);
#endif

    SDIAS_TIMEOUT_TASK:
#ifdef HWC_LogValue1
      HWC_LogValue1(this, "@00A4 (SdiasManager::LogSDOErrorInfo) SDO Error 0x{0}: Timeout of task", (0-OSRetVal)$UDINT);
#endif

    SDIAS_RESPONSE_BUFFER_TOO_SMALL:
#ifdef HWC_LogValue1
      HWC_LogValue1(this, "@00A5 (SdiasManager::LogSDOErrorInfo) SDO Error 0x{0}: Response buffer too small", (0-OSRetVal)$UDINT);
#endif

    SDIAS_TIMEOUT_SDO_RESPONSE:
#ifdef HWC_LogValue1
      HWC_LogValue1(this, "@00A6 (SdiasManager::LogSDOErrorInfo) SDO Error 0x{0}: Timeout SDO response", (0-OSRetVal)$UDINT);
#endif

    SDIAS_OUT_OF_HANDLES:
#ifdef HWC_LogValue1
      HWC_LogValue1(this, "@00A7 (SdiasManager::LogSDOErrorInfo) SDO Error 0x{0}: Out of handles", (0-OSRetVal)$UDINT);
#endif

    SDIAS_INVALID_PARAM_DATA_LENGTH:
#ifdef HWC_LogValue1
      HWC_LogValue1(this, "@00A8 (SdiasManager::LogSDOErrorInfo) SDO Error 0x{0}: Invalid length of data bytes", (0-OSRetVal)$UDINT);
#endif

    SDIAS_INVALID_PARAM_DATA_BUFFER:
#ifdef HWC_LogValue1
      HWC_LogValue1(this, "@00A9 (SdiasManager::LogSDOErrorInfo) SDO Error 0x{0}: Invalid data buffer", (0-OSRetVal)$UDINT);
#endif

    SDIAS_INVALID_PARAM_SDO_HANDLE:
#ifdef HWC_LogValue1
      HWC_LogValue1(this, "@00AA (SdiasManager::LogSDOErrorInfo) SDO Error 0x{0}: Invalid SDO handle", (0-OSRetVal)$UDINT);
#endif

    SDIAS_INVALID_PARAM_NODE:
#ifdef HWC_LogValue1
      HWC_LogValue1(this, "@00AB (SdiasManager::LogSDOErrorInfo) SDO Error 0x{0}: Invalid node handle", (0-OSRetVal)$UDINT);
#endif

    SDIAS_GLOBAL_ERROR:
#ifdef HWC_LogValue1
      HWC_LogValue1(this, "@00AC (SdiasManager::LogSDOErrorInfo) SDO Error 0x{0}: General Error of SDIAS Manager", (0-OSRetVal)$UDINT);
#endif

    SDIAS_INVALID_MANAGER:
#ifdef HWC_LogValue1
      HWC_LogValue1(this, "@00AD (SdiasManager::LogSDOErrorInfo) SDO Error 0x{0}: SDIAS Manager not found", (0-OSRetVal)$UDINT);
#endif

    SDIAS_SENDING_SDO_REQUEST_FAILED:
#ifdef HWC_LogValue1
      HWC_LogValue1(this, "@00AE (SdiasManager::LogSDOErrorInfo) SDO Error 0x{0}: Sending SDO request failed", (0-OSRetVal)$UDINT);
#endif

    SDIAS_RECEIVING_SDO_RESPONSE_FAILED:
#ifdef HWC_LogValue1
      HWC_LogValue1(this, "@00AF (SdiasManager::LogSDOErrorInfo) SDO Error 0x{0}: Receiving SDO response failed", (0-OSRetVal)$UDINT);
#endif

    SDIAS_MANAGER_GLOBAL_ERROR:
#ifdef HWC_LogValue1
      HWC_LogValue1(this, "@00B0 (SdiasManager::LogSDOErrorInfo) SDO Error 0x{0}: General Error of SDIAS Manager (like communication problems to client)", (0-OSRetVal)$UDINT);
#endif

    SDIAS_INTERNAL_ERROR:
#ifdef HWC_LogValue1
      HWC_LogValue1(this, "@00B1 (SdiasManager::LogSDOErrorInfo) SDO Error 0x{0}: Internal error", (0-OSRetVal)$UDINT);
#endif

  else
#ifdef HWC_LogValue1
    HWC_LogValue1(this, "@00B2 (SdiasManager::LogSDOErrorInfo) SDO Error 0x{0}: Unknown Error", (0-OSRetVal)$UDINT);
#endif
  end_case;

END_FUNCTION

FUNCTION VIRTUAL SdiasManager::CheckAccess
	VAR_INPUT
		bsStateByte 	: t_SDIAS_StateByte;
		sdRequired 	: DINT;
		sdPlace 	: DINT;
		pCrashThisTime 	: ^USINT;
		pCrashMessage 	: ^CHAR;
	END_VAR
	VAR_OUTPUT
		usRetryCounter 	: USINT;
	END_VAR

  // increase retrycounter if retries occured on the access
  usRetryCounter := bsStateByte SHR 5;

  // check if the access failed
  if sdRequired & (bsStateByte.AccessFailed = TRUE) then
    ModuleObjInfo[sdPlace].pThis^.ClassState := _RequiredError;
    RequiredPlace := sdPlace;
    CyclicMsgMarker.PostIt.RequiredError := TRUE;
    ClassState := _RequiredError;
    ErrorInitStep := InitSSW;
    InitSSW := _PrepareError;

    pCrashThisTime^ := 2;

    _strcpy(dest:=pCrashMessage, src:="Access to a required SDIAS Module failed");
  end_if;

END_FUNCTION

FUNCTION VIRTUAL SdiasManager::PostRtMessages

  // if there are some messages to post, post them (the methods in the brackets are not the actual, but the methods were the error occured)
  if CyclicMsgMarker.PostIt then
    if CyclicMsgMarker.PostIt.IsoReadRunFailed then
#ifdef HWC_LogError
      HWC_LogError(this, "@00B3 (SdiasManager::RtWork) Error changing the run state of the isochronous read access!");
#endif
    end_if;

    if CyclicMsgMarker.PostIt.IsoWriteRunFailed then
#ifdef HWC_LogError
      HWC_LogError(this, "@00B4 (SdiasManager::RtWork) Error changing the run state of the isochronous write access!");
#endif
    end_if;

    if CyclicMsgMarker.PostIt.RequiredError then
#ifdef HWC_LogValue1
      HWC_LogValue1(this, "@00B5 (SdiasManager::RtWork) Required Error at SDIAS Place 0x{0}", RequiredPlace$UDINT);
#endif
    end_if;

    if CyclicMsgMarker.PostIt.ForwardRequiredErrorFailed then
#ifdef HWC_LogError
      HWC_LogError(this, "@00B6 (SdiasManager::RtWork) Failed to set required error to BusInterface");
#endif
    end_if;

    if CyclicMsgMarker.PostIt.ToggleErrorWrTask & (CyclicMsgMarker.AlreadyPosted.ToggleErrorWrTask = FALSE) then
#ifdef HWC_LogError
      HWC_LogError(this, "@00B7 (SdiasManager::RtWork) [SL] Error at toggle bit of iso write task of SDIAS");
#endif
      CyclicMsgMarker.AlreadyPosted.ToggleErrorWrTask := TRUE;
    end_if;

    if CyclicMsgMarker.PostIt.ToggleErrorRdTask & (CyclicMsgMarker.AlreadyPosted.ToggleErrorRdTask = FALSE) then
#ifdef HWC_LogError
      HWC_LogError(this, "@00B8 (SdiasManager::RtWork) [SL] Error at toggle bit of iso read task of SDIAS");
#endif
      CyclicMsgMarker.AlreadyPosted.ToggleErrorRdTask := TRUE;
    end_if;

    if CyclicMsgMarker.PostIt.ErrorWrTask & (CyclicMsgMarker.AlreadyPosted.ErrorWrTask = FALSE) then
#ifdef HWC_LogValue1
      HWC_LogValue1(this, "@00B9 (SdiasManager::RtWork) [SL] Error at iso write task of SDIAS 0x{0}", (WriteTaskInfo.pReadData^.ErrorInfoFlags AND SDIAS_ERROR_INFO_MASK));
#endif
      CyclicMsgMarker.AlreadyPosted.ErrorWrTask := TRUE;
    end_if;

    if CyclicMsgMarker.PostIt.ErrorRdTask & (CyclicMsgMarker.AlreadyPosted.ErrorRdTask = FALSE) then
#ifdef HWC_LogValue1
      HWC_LogValue1(this, "@00BA (SdiasManager::RtWork) [SL] Error at iso read task of SDIAS 0x{0}", (ReadTaskInfo.pReadData^.ErrorInfoFlags AND SDIAS_ERROR_INFO_MASK));
#endif
      CyclicMsgMarker.AlreadyPosted.ErrorRdTask := TRUE;
    end_if;

    if CyclicMsgMarker.PostIt.GetRdInfoFailed & (CyclicMsgMarker.AlreadyPosted.GetRdInfoFailed = FALSE) then
#ifdef HWC_LogError
      HWC_LogError(this, "@00BB (SdiasManager::RtWork) [SL] Error fetching iso read task info from OS");
#endif
      CyclicMsgMarker.AlreadyPosted.GetRdInfoFailed := TRUE;
    end_if;

    if CyclicMsgMarker.PostIt.GetWrInfoFailed & (CyclicMsgMarker.AlreadyPosted.GetWrInfoFailed = FALSE) then
#ifdef HWC_LogError
      HWC_LogError(this, "@00BC (SdiasManager::RtWork) [SL] Error fetching iso write task info from OS");
#endif
      CyclicMsgMarker.AlreadyPosted.GetWrInfoFailed := TRUE;
    end_if;

    if CyclicMsgMarker.PostIt.SetSyncFailed & (CyclicMsgMarker.AlreadyPosted.SetSyncFailed = FALSE) then
#ifdef HWC_LogError
      HWC_LogError(this, "@00BD (SdiasManager::RtWork) [SL] Failed to set sync out of pll");
#endif
      CyclicMsgMarker.AlreadyPosted.SetSyncFailed := TRUE;
    end_if;

    if CyclicMsgMarker.PostIt.GetFrameCounterFailed & (CyclicMsgMarker.AlreadyPosted.GetFrameCounterFailed = FALSE) then
#ifdef HWC_LogError
      HWC_LogError(this, "@00BE (SdiasManager::RtWork) [SL] Failed to get the frame counter info via OS interface");
#endif
      CyclicMsgMarker.AlreadyPosted.SetSyncFailed := TRUE;
    end_if;

    if CyclicMsgMarker.PostIt.WrTaskNotFinished & (CyclicMsgMarker.AlreadyPosted.WrTaskNotFinished = FALSE) then
#ifdef HWC_LogError
      HWC_LogError(this, "@00BF (SdiasManager::RtWork) [SL] Iso write task of SDIAS hasn't been completed");
#endif
      CyclicMsgMarker.AlreadyPosted.WrTaskNotFinished := TRUE;
    end_if;

    if CyclicMsgMarker.PostIt.WrTaskInterruptedByRdTask & (CyclicMsgMarker.AlreadyPosted.WrTaskInterruptedByRdTask = FALSE) then
#ifdef HWC_LogError
      HWC_LogError(this, "@00C0 (SdiasManager::RtWork) [SL] Iso write task of SDIAS has been interrupted by read task");
#endif
      CyclicMsgMarker.AlreadyPosted.WrTaskInterruptedByRdTask := TRUE;
    end_if;

    if CyclicMsgMarker.PostIt.RdTaskNotFinished & (CyclicMsgMarker.AlreadyPosted.RdTaskNotFinished = FALSE) then
      // this happens on local SDIAS:
      //  - if the iso startpoint is too high and the SDIAS read task can't finish before the next RT
      //
      // on SDIAS via VARAN:
      //  - VARAN iso startpoint too low or SDIAS read task load too high => task is not finished when the data is fetched via VARAN
#ifdef HWC_LogError
      HWC_LogError(this, "@00C1 (SdiasManager::RtWork) [SL] Iso read task of SDIAS hasn't been completed! Check setting of IsoStartPoint and cycle time!");
#endif
      CyclicMsgMarker.AlreadyPosted.RdTaskNotFinished := TRUE;
    end_if;
    if CyclicMsgMarker.PostIt.RdTaskNoEvent & (CyclicMsgMarker.AlreadyPosted.RdTaskNoEvent = FALSE) then
      // this happens on local SDIAS:
      //  - the RT takes too long and the SDIAS read task doesn't even start
      //
      // on SDIAS via VARAN:
      //  - VARAN iso startpoint or VARAN load too high => SDIAS read task doesn't even start
#ifdef HWC_LogError
      HWC_LogError(this, "@00C2 (SdiasManager::RtWork) [SL] Iso read task of SDIAS hasn't been started! Check setting of IsoStartPoint and cycle time!");
#endif
      CyclicMsgMarker.AlreadyPosted.RdTaskNoEvent := TRUE;
    end_if;

    if CyclicMsgMarker.PostIt.TaskInfoRunFailed then
#ifdef HWC_LogError
      HWC_LogError(this, "@00C3 (SdiasManager::RtWork) Error changing the run state of the isochronous read access to get the task info!");
#endif
    end_if;

    if CyclicMsgMarker.PostIt.IsoConfigWrTaskConfigFailed then
#ifdef HWC_LogError
      HWC_LogError(this, "@00C4 (SdiasManager::RtWork) Error starting isochronous configuration write access with single for task config!");
#endif
    end_if;

    if CyclicMsgMarker.PostIt.IsoConfigWrTriggerUnitFailed then
#ifdef HWC_LogError
      HWC_LogError(this, "@00C5 (SdiasManager::RtWork) Error starting isochronous configuration write access with single for trigger unit settings!");
#endif
    end_if;

    if CyclicMsgMarker.PostIt.IsoConfigWrChangeFailed then
#ifdef HWC_LogError
      HWC_LogError(this, "@00C6 (SdiasManager::RtWork) Failed to change the isochronous configuration write access!");
#endif
    end_if;

    if CyclicMsgMarker.PostIt.IsoTaskConfigFailed then
#ifdef HWC_LogError
      HWC_LogError(this, "@00C7 (SdiasManager::RtWork) Failed to set the iso read start config via OS interface!");
#endif
    end_if;

    if CyclicMsgMarker.PostIt.IsoTriggerUnitConfigFailed then
#ifdef HWC_LogError
      HWC_LogError(this, "@00C8 (SdiasManager::RtWork) Failed to set the trigger unit config via OS interface!");
#endif
    end_if;

    if CyclicMsgMarker.PostIt.IsoConfigWrChange2Failed then
#ifdef HWC_LogError
      HWC_LogError(this, "@00C9 (SdiasManager::RtWork) Error changing isochronous configuration write access for sync injection!");
#endif
    end_if;

    if CyclicMsgMarker.PostIt.IsoConfigWrSyncInjFailed then
#ifdef HWC_LogError
      HWC_LogError(this, "@00CA (SdiasManager::RtWork) Error starting isochronous configuration write access with single RUN for sync injection!");
#endif
    end_if;

    if CyclicMsgMarker.PostIt.IsoSyncInjFailed then
#ifdef HWC_LogError
      HWC_LogError(this, "@00CB (SdiasManager::RtWork) Failed to set the sync injection config via OS interface!");
#endif
    end_if;

    if CyclicMsgMarker.PostIt.SetOnlineStateFailed then
#ifdef HWC_LogError
      HWC_LogError(this, "@00CC (SdiasManager::RtWork) Failed to set the Online state!");
#endif
    end_if;

    CyclicMsgMarker.PostIt := 0;
  end_if;

END_FUNCTION

FUNCTION VIRTUAL SdiasManager::ChangeDynAccess
	VAR_INPUT
		AccessHandle 	: UDINT;
		NewOffset 	: HDINT;
		NewLength 	: UDINT;
	END_VAR
	VAR_OUTPUT
		Success 	: BOOL;
	END_VAR
  VAR
  	pAccess           : ^t_AccessElement;
    pControlStruct    : ^t_SDIAS_ControlStructDynamic;
    pControlStructFar : ^t_SDIAS_ControlStructDynamicFar;
    usBlockNo1k       : USINT;
    hiModAddr0        : HINT;
  END_VAR

  Success := FALSE;

  // check if valid handle
  if AccessHandle then
    pAccess := AccessHandle$^t_AccessElement;

    if (pAccess^.eAccessType = _ReadDynamic) | (pAccess^.eAccessType = _WriteDynamic) then
      if pAccess^.bIsFarAcc then
        pControlStructFar := (pAccess^.ppControlByte^)$^t_SDIAS_ControlStructDynamicFar;
        if pControlStructFar then
          if pAccess^.eAccessType = _ReadDynamic then
            if NewLength <> SDIAS_UNCHANGED_DYNAMIC_PARA then
              if NewLength > SDIAS_MAX_SIZE_FAR_MEM_ACCESS then
                return;
              else
                pControlStructFar^.usLengthRd := NewLength$USINT;
              end_if;
            end_if;
            if NewOffset <> SDIAS_UNCHANGED_DYNAMIC_PARA then
              usBlockNo1k     := to_usint(NewOffset shr 10);
              hiModAddr0     := (NewOffset AND 16#3FF)$HINT + (pAccess^.usPlace shl 10);
              pControlStructFar^.hiOffsetRd := hiModAddr0;
              pControlStructFar^.hiOffsetWr := usBlockNo1k;
            end_if;
            Success := TRUE;

          else // _WriteDynamic
            if NewLength <> SDIAS_UNCHANGED_DYNAMIC_PARA then
              if NewLength > SDIAS_MAX_SIZE_FAR_MEM_ACCESS then
                return;
              else
                pControlStructFar^.usLengthWr := NewLength$USINT;
              end_if;
              if NewOffset <> SDIAS_UNCHANGED_DYNAMIC_PARA then
                usBlockNo1k     := to_usint(NewOffset shr 10);
                hiModAddr0     := (NewOffset AND 16#3FF)$HINT + (pAccess^.usPlace shl 10);
                pControlStructFar^.hiOffsetWr := hiModAddr0;
                pControlStructFar^.hiOffsetRd := usBlockNo1k;
              end_if;
              Success := TRUE;

           end_if;
          end_if;
        end_if;
      else
        pControlStruct := (pAccess^.ppControlByte^)$^t_SDIAS_ControlStructDynamic;

        if pControlStruct then
          if NewOffset <> SDIAS_UNCHANGED_DYNAMIC_PARA then
            pControlStruct^.hiOffset := NewOffset$HINT + (pAccess^.usPlace shl 10);
          end_if;

          if NewLength <> SDIAS_UNCHANGED_DYNAMIC_PARA then
            pControlStruct^.usLength := NewLength$USINT;
          end_if;

          Success := TRUE;
        end_if;
      end_if;
    end_if;
  end_if;

END_FUNCTION

FUNCTION VIRTUAL SdiasManager::CreateAndModifyIsoDOs
  VAR
    dataUPDATEDO          : t_UpdateDOCfg;
    dataADDDO             : t_AddDOCfg;
  	tempCmd               : CmdStruct;
    _result               : results;
  END_VAR

  // initialize the data for the task config in realtime

  // set the task duration limit
  ISOTaskConfig.TaskDurationTimeout_us := (ud_BusTime_ns / 1000)$UINT;

  // start address of iso read list
  ISOTaskConfig.Config := gcMapping_Informations[IsoRdList].StartAddress;

  // we want to use the start configuration => enable it
  ISOTaskConfig.Config.SynchronizedStartEnable := TRUE;

  // initialize the data for the trigger unit setup for later use
  ISOTriggerUnitSetup.TaskSelect := 0;
  ISOTriggerUnitSetup.TaskSelect.IsoWrite := TRUE;
  ISOTriggerUnitSetup.TaskSelect.IsoRead  := TRUE;

  ISOTriggerUnitSetup.StartAddress := gcMapping_Informations[IsoWrPayload].StartAddress - SDIAS_TRIGGER_UNIT_BYTE_SIZE;
  ISOTriggerUnitSetup.StartAddress.UnitEnable := TRUE;

  if ConnectionType = SDIAS_CON_VIA_VARAN_uC then

    if b_IsoDOsCreated = FALSE then

#ifndef SDIAS_DEACTIVATE_TASK_CHECKS
      // DO for Task Infos (start at task 1 = read task)
      TaskInfoDO.Offset := SDIAS_OFFSET_TASK_INFO_1;
      TaskInfoDO.Length := sizeof(t_TaskInfoReadData);

      dataADDDO.Priority            := _BUS_IF_ISO_MOVE;
      dataADDDO.RdWr                := _BUS_IF_READ;
      dataADDDO.ud_addressoff_read  := TaskInfoDO.Offset;
      dataADDDO.ui_length_read      := TaskInfoDO.Length;
      dataADDDO.b_UseLocalCopy      := TRUE;

      tempCmd.uiCmd     := _BUS_IF_ADD_DO;
      tempCmd.aPara[0]  := (#dataADDDO)$DINT;

      ToBusInterface.NewInst(pPara:=#tempCmd, pResult:=#_result);
      if _result.aData[0]$t_BusIFRetvalErrorcode = _BUS_IF_RETVAL_OK then
        TaskInfoDO.Handle        := _result.aData$t_AddDORet.Handle;
        TaskInfoDO.pData         := _result.aData$t_AddDORet.pDataRead;
        TaskInfoDO.AccessHandle  := _result.aData$t_AddDORet.AccessHandle;

        // the parameter is overwritten with the DPRAM adress if the pData points to local memory
        TaskInfoDO.pDataDPRAM := dataADDDO.ud_addressoff_read$pVoid;
      else
#ifdef HWC_LogError
        HWC_LogError(this, "@00CD (SdiasManager::CreateAndModifyIsoDOs) Failed to add DO for the task info");
#endif
        InitError := _CreateDOFailed;
      end_if;
#endif

      // DO to enable read task in realtime before going to operational state
      dataADDDO.Priority            := _BUS_IF_ISO_MOVE;
      dataADDDO.RdWr                := _BUS_IF_WRITE;
      dataADDDO.ud_addressoff_write := SDIAS_OFFSET_TASK_CONFIG_1;
      dataADDDO.ui_length_write     := sizeof(t_TaskConfig);
      dataADDDO.b_UseLocalCopy      := TRUE;

      tempCmd.uiCmd     := _BUS_IF_ADD_DO;
      tempCmd.aPara[0]  := (#dataADDDO)$DINT;

      ToBusInterface.NewInst(pPara:=#tempCmd, pResult:=#_result);
      if _result.aData[0]$t_BusIFRetvalErrorcode = _BUS_IF_RETVAL_OK then
        ISOConfigWrDO.Handle        := _result.aData$t_AddDORet.Handle;
        ISOConfigWrDO.pData         := _result.aData$t_AddDORet.pDataWrite;
        ISOConfigWrDO.AccessHandle  := _result.aData$t_AddDORet.AccessHandle;

        // the parameter is overwritten with the DPRAM adress if the pData points to local memory
        ISOConfigWrDO.pDataDPRAM := dataADDDO.ud_addressoff_write$pVoid;

        // the first thing we write is the task config
        ISOConfigWrDO.pData^$t_TaskConfig := ISOTaskConfig;
      else
#ifdef HWC_LogError
        HWC_LogError(this, "@00CE (SdiasManager::CreateAndModifyIsoDOs) Failed to add DO for starting the iso read task");
#endif
        InitError := _CreateDOFailed;
      end_if;

      // recalculate payload size for accessing the payload

      AddBroadCastAccessesToList();

      // take our special access usage and add the usage according to the µC as well as 2 bytes for the trigger unit activation
      ISOWriteDO.Length += gcMapping_Informations[IsoWrPayload].ActUsage + SDIAS_TRIGGER_UNIT_BYTE_SIZE;

      // take our special access usage and add the usage according to the µC
      ISOReadDO.Length  += gcMapping_Informations[IsoRdPayload].ActUsage;

      // since we get the status info extra => skip the status byte of watchdog + status byte of write task info + write task info + status byte of read task info + read task info
      ISOReadDO.Length  -= sizeof(t_SDIAS_StateByte) + sizeof(t_SDIAS_StateByte) + sizeof(t_TaskInfoData.Handshake) + sizeof(t_TaskInfoData.DurationTime) + sizeof(t_TaskInfoData.ExecutionTime)
                                                     + sizeof(t_SDIAS_StateByte) + sizeof(t_TaskInfoData.Handshake) + sizeof(t_TaskInfoData.DurationTime) + sizeof(t_TaskInfoData.ExecutionTime);

      // Long DO for Read Data
      dataADDDO.Priority            := _BUS_IF_ISO_MOVE;
      dataADDDO.RdWr                := _BUS_IF_READ;
      dataADDDO.ud_addressoff_read  := 0;
      dataADDDO.ui_length_read      := ISOReadDO.Length;
      dataADDDO.b_UseLocalCopy      := TRUE;

      tempCmd.uiCmd     := _BUS_IF_ADD_DO;
      tempCmd.aPara[0]  := (#dataADDDO)$DINT;

      ToBusInterface.NewInst(pPara:=#tempCmd, pResult:=#_result);
      if _result.aData[0]$t_BusIFRetvalErrorcode = _BUS_IF_RETVAL_OK then
        ISOReadDO.Handle        := _result.aData$t_AddDORet.Handle;
        ISOReadDO.pData         := _result.aData$t_AddDORet.pDataRead;
        ISOReadDO.AccessHandle  := _result.aData$t_AddDORet.AccessHandle;

        // the parameter is overwritten with the DPRAM adress if the pData points to local memory
        ISOReadDO.pDataDPRAM := dataADDDO.ud_addressoff_read$pVoid;
      else
#ifdef HWC_LogError
        HWC_LogError(this, "@00CF (SdiasManager::CreateAndModifyIsoDOs) Failed to add long DO for the isochronous read data");
#endif
        InitError := _CreateDOFailed;
      end_if;

      // Long DO for Write Data
      dataADDDO.Priority            := _BUS_IF_ISO_MOVE;
      dataADDDO.RdWr                := _BUS_IF_WRITE;
      dataADDDO.ud_addressoff_write := 0;
      dataADDDO.ui_length_write     := ISOWriteDO.Length;
      dataADDDO.b_UseLocalCopy      := TRUE;

      tempCmd.uiCmd     := _BUS_IF_ADD_DO;
      tempCmd.aPara[0]  := (#dataADDDO)$DINT;

      ToBusInterface.NewInst(pPara:=#tempCmd, pResult:=#_result);
      if _result.aData[0]$t_BusIFRetvalErrorcode = _BUS_IF_RETVAL_OK then
        ISOWriteDO.Handle       := _result.aData$t_AddDORet.Handle;
        ISOWriteDO.pData        := _result.aData$t_AddDORet.pDataWrite;
        ISOWriteDO.AccessHandle := _result.aData$t_AddDORet.AccessHandle;

        // the parameter is overwritten with the DPRAM adress if the pData points to local memory
        ISOWriteDO.pDataDPRAM := dataADDDO.ud_addressoff_write$pVoid;
      else
#ifdef HWC_LogError
        HWC_LogError(this, "@00D0 (SdiasManager::CreateAndModifyIsoDOs) Failed to add long DO for the isochronous write data");
#endif
        InitError := _CreateDOFailed;
      end_if;

      // reset data objects (calculate retry timeout) is done before the runstate is set

      //Save length of ISO Read and ISO Write DO, will later be used to check if the length is correct when there is a reconnect
      //It can happen that there is only 1 module at the first connect and at the second connect there are 5 SDIAS module behind the VI02x
      //We save the created length here and check it later if the length is ok
      sDOLengthsFirstConnect.udISOReadLength :=     ISOReadDO.Length;
      sDOLengthsFirstConnect.udISOWriteLength :=    ISOWriteDO.Length;
      sDOLengthsFirstConnect.udISOReadActUsage :=   gcMapping_Informations[IsoRdPayload].ActUsage;
      sDOLengthsFirstConnect.udISOWriteActUsage :=  gcMapping_Informations[IsoWrPayload].ActUsage;

      if InitError <> _CreateDOFailed then
        b_IsoDOsCreated := TRUE;
        b_IsoDOsJustCreated := TRUE;
      end_if;
    end_if;
  end_if;

  // first we need to check out where our payload is stored and if it got the right size to access the right memory
  if gcMapping_Informations[IsoWrPayload].StartAddress then
    // modify if connected via VARAN
    if ConnectionType = SDIAS_CON_VIA_VARAN_uC then

                                                                                 // trigger unit is not actually part of the usage
      ISOWriteDO.Offset := gcMapping_Informations[IsoWrPayload].StartAddress - SDIAS_TRIGGER_UNIT_BYTE_SIZE; // the trigger unit starts earlier

      ISOWriteDO.pData^$UINT := ISOWriteDO.Length - SDIAS_TRIGGER_UNIT_BYTE_SIZE; // trigger unit itself is not part of the payload data size

      dataUPDATEDO.Handle               := ISOWriteDO.Handle;
      dataUPDATEDO.ud_addressoff_write  := ISOWriteDO.Offset;
      dataUPDATEDO.ud_length_write      := ISOWriteDO.Length;

      tempCmd.uiCmd         := _BUS_IF_UPDATE_DO;
      tempCmd.aPara[0]      := (#dataUPDATEDO)$DINT;

      ToBusInterface.NewInst(pPara:=#tempCmd, pResult:=#_result);
      if _result.aData[0]$t_BusIFRetvalErrorcode <> _BUS_IF_RETVAL_OK then
#ifdef HWC_LogError
        HWC_LogError(this, "@00D3 (SdiasManager::CreateAndModifyIsoDOs) Failed to change isochronous write access! Unable to continue with Initialisation!");
#endif
        ClassState := _ManagerError;
        ErrorInitStep := InitSSW;
        InitSSW := _PrepareError;
        return;
      end_if;
    else
      // create if connected locally

      // Long DO for Write Data

      AddBroadCastAccessesToList();

      // take our special access usage and add the usage according to the µC as well as 2 bytes for the trigger unit activation
      ISOWriteDO.Length += gcMapping_Informations[IsoWrPayload].ActUsage + SDIAS_TRIGGER_UNIT_BYTE_SIZE;

      ISOWriteDO.Offset := gcMapping_Informations[IsoWrPayload].StartAddress - SDIAS_TRIGGER_UNIT_BYTE_SIZE; // the trigger unit starts earlier

      dataADDDO.Priority            := _BUS_IF_ISO_MOVE;
      dataADDDO.RdWr                := _BUS_IF_WRITE;
      dataADDDO.ud_addressoff_write := ISOWriteDO.Offset;
      dataADDDO.ui_length_write     := ISOWriteDO.Length;
      dataADDDO.ud_addressoff_read  := 0;
      dataADDDO.ui_length_read      := 0;
      dataADDDO.b_UseLocalCopy      := TRUE;

      tempCmd.uiCmd     := _BUS_IF_ADD_DO;
      tempCmd.aPara[0]  := (#dataADDDO)$DINT;

      ToBusInterface.NewInst(pPara:=#tempCmd, pResult:=#_result);
      if _result.aData[0]$t_BusIFRetvalErrorcode = _BUS_IF_RETVAL_OK then
        ISOWriteDO.Handle       := _result.aData$t_AddDORet.Handle;
        ISOWriteDO.pData        := _result.aData$t_AddDORet.pDataWrite;
        ISOWriteDO.AccessHandle := _result.aData$t_AddDORet.AccessHandle;

        // initialize the trigger unit
        ISOWriteDO.pData^$UINT := ISOWriteDO.Length - SDIAS_TRIGGER_UNIT_BYTE_SIZE;

        // the parameter is overwritten with the DPRAM adress if the pData points to local memory
        ISOWriteDO.pDataDPRAM := dataADDDO.ud_addressoff_write$pVoid;
      else
#ifdef HWC_LogError
        HWC_LogError(this, "@00D0 (SdiasManager::CreateAndModifyIsoDOs) Failed to add long DO for the isochronous write data");
#endif
        InitError := _CreateDOFailed;
      end_if;
    end_if;
  end_if;

  if gcMapping_Informations[IsoRdPayload].StartAddress then
    // modify if connected via VARAN
    if ConnectionType = SDIAS_CON_VIA_VARAN_uC then
      ISOReadDO.Offset := gcMapping_Informations[IsoRdPayload].StartAddress;

      // since we get the status info extra => skip the status byte of watchdog + status byte of write task info + write task info + status byte of read task info + read task info
      ISOReadDO.Offset += sizeof(t_SDIAS_StateByte) + sizeof(t_SDIAS_StateByte) + sizeof(t_TaskInfoData.Handshake) + sizeof(t_TaskInfoData.DurationTime) + sizeof(t_TaskInfoData.ExecutionTime)
                                                    + sizeof(t_SDIAS_StateByte) + sizeof(t_TaskInfoData.Handshake) + sizeof(t_TaskInfoData.DurationTime) + sizeof(t_TaskInfoData.ExecutionTime);

      dataUPDATEDO.Handle               := ISOReadDO.Handle;
      dataUPDATEDO.ud_addressoff_read   := ISOReadDO.Offset;
      dataUPDATEDO.ud_length_read       := ISOReadDO.Length;

      tempCmd.uiCmd         := _BUS_IF_UPDATE_DO;
      tempCmd.aPara[0]      := (#dataUPDATEDO)$DINT;

      ToBusInterface.NewInst(pPara:=#tempCmd, pResult:=#_result);
      if _result.aData[0]$t_BusIFRetvalErrorcode <> _BUS_IF_RETVAL_OK then
#ifdef HWC_LogError
        HWC_LogError(this, "@00D4 (SdiasManager::CreateAndModifyIsoDOs) Failed to change isochronous read access! Unable to continue with Initialisation!");
#endif
        ClassState := _ManagerError;
        ErrorInitStep := InitSSW;
        InitSSW := _PrepareError;
        return;
      end_if;
    else
      // create if connected locally

      // Long DO for Read Data

      // take our special access usage and add the usage according to the µC
      ISOReadDO.Length  += gcMapping_Informations[IsoRdPayload].ActUsage;

      ISOReadDO.Offset := gcMapping_Informations[IsoRdPayload].StartAddress;

      dataADDDO.Priority            := _BUS_IF_ISO_MOVE;
      dataADDDO.RdWr                := _BUS_IF_READ;
      dataADDDO.ud_addressoff_read  := ISOReadDO.Offset;
      dataADDDO.ui_length_read      := ISOReadDO.Length;
      dataADDDO.ud_addressoff_write := 0;
      dataADDDO.ui_length_write     := 0;
      dataADDDO.b_UseLocalCopy      := TRUE;

      tempCmd.uiCmd     := _BUS_IF_ADD_DO;
      tempCmd.aPara[0]  := (#dataADDDO)$DINT;

      ToBusInterface.NewInst(pPara:=#tempCmd, pResult:=#_result);
      if _result.aData[0]$t_BusIFRetvalErrorcode = _BUS_IF_RETVAL_OK then
        ISOReadDO.Handle        := _result.aData$t_AddDORet.Handle;
        ISOReadDO.pData         := _result.aData$t_AddDORet.pDataRead;
        ISOReadDO.AccessHandle  := _result.aData$t_AddDORet.AccessHandle;

        // the parameter is overwritten with the DPRAM adress if the pData points to local memory
        ISOReadDO.pDataDPRAM := dataADDDO.ud_addressoff_read$pVoid;
      else
#ifdef HWC_LogError
        HWC_LogError(this, "@00CF (SdiasManager::CreateAndModifyIsoDOs) Failed to add long DO for the isochronous read data");
#endif
        InitError := _CreateDOFailed;
      end_if;
    end_if;
  end_if;

END_FUNCTION

FUNCTION VIRTUAL SdiasManager::IsDeviceBitSet
	VAR_INPUT
		pDeviceBitMap 	: ^BDINT;
		Place 	: UDINT;
	END_VAR
	VAR_OUTPUT
		bIsSet 	: BOOL;
	END_VAR

  if Place >= 32 then
    Place -= 32;
    pDeviceBitmap += 4;
  end_if;
  bIsSet := ((pDeviceBitmap^ SHR Place) AND 1)$BOOL;

END_FUNCTION

FUNCTION VIRTUAL SdiasManager::DisableBus
  VAR
    dataSETRUNSTATE     : t_SetRunStateCfg;
  	tempCmd             : CmdStruct;
    _result             : results;
    dataUPDATEDO        : t_UpdateDOCfg;
    aProperties         : ARRAY [0..4] OF SDM_PROPERTY_VALUE_PAIR;
    SyncInjectionCfg    : t_SyncInjectionCfg;
  END_VAR

  // we select the read task for sync, there are no sync task trigger losses allowed and we disable the sync injection
  SyncInjectionCfg := 16#02;

  if ConnectionType = SDIAS_CON_VIA_VARAN_uC then
    // change config DO => change trigger unit settings (also use trigger unit for read task)
    ISOConfigWrDO.Offset := SDIAS_OFFSET_SYNC_INJECTION_CFG;
    ISOConfigWrDO.Length := sizeof(t_SyncInjectionCfg);

    dataUPDATEDO.Handle               := ISOConfigWrDO.Handle;
    dataUPDATEDO.ud_addressoff_write  := ISOConfigWrDO.Offset;
    dataUPDATEDO.ud_length_write      := ISOConfigWrDO.Length;

    tempCmd.uiCmd         := _BUS_IF_UPDATE_DO;
    tempCmd.aPara[0]      := (#dataUPDATEDO)$DINT;

    ToBusInterface.NewInst(pPara:=#tempCmd, pResult:=#_result);

    if _result.aData[0]$t_BusIFRetvalErrorcode <> _BUS_IF_RETVAL_OK then
      // remember the log message and write it in cyclic priority to avoid a rt runtime error
      CyclicMsgMarker.PostIt.IsoConfigWrChange2Failed := TRUE;
    else
      // use the sync injection data
      ISOConfigWrDO.pData^$t_SyncInjectionCfg := SyncInjectionCfg;
    end_if;

    dataSETRUNSTATE.NewRunState := _BUS_IF_RUN_STATE_SINGLE_RUN;
    tempCmd.uiCmd               := _BUS_IF_SET_RUN_STATE;
    tempCmd.aPara[0]            := (#dataSETRUNSTATE)$DINT;

    dataSETRUNSTATE.Handle      := ISOConfigWrDO.Handle;

    ToBusInterface.NewInst(pPara:=#tempCmd, pResult:=#_result);

    if _result.aData[0]$t_BusIFRetvalErrorcode <> _BUS_IF_RETVAL_OK then
      // remember the log message and write it in cyclic priority to avoid a rt runtime error
      CyclicMsgMarker.PostIt.IsoConfigWrSyncInjFailed := TRUE;
    end_if;
  else
    aProperties[0].udPropertyId     := SDM_PROP_SYNC_INJECTION_CONFIG;
    aProperties[0].udPropertyValue  := SyncInjectionCfg;

    if SDIAS_iSetNodeProperties(hNodeHandle         := udNodeHandle
                              , udPropertyCount     := 1
                              , psPropertyValuePairs:= #aProperties[0]
                              ) <> SDIAS_OK then
      // remember the log message and write it in cyclic priority to avoid a rt runtime error
      CyclicMsgMarker.PostIt.IsoSyncInjFailed := TRUE;
    end_if;
  end_if;

  // general settings needed for all DOs
  dataSETRUNSTATE.NewRunState := _BUS_IF_RUN_STATE_NO_RUN;
  tempCmd.uiCmd         := _BUS_IF_SET_RUN_STATE;
  tempCmd.aPara[0]      := (#dataSETRUNSTATE)$DINT;

#ifndef SDIAS_DEACTIVATE_TASK_CHECKS
  if ConnectionType = SDIAS_CON_VIA_VARAN_uC then
    // set runstate of taskinfo read
    dataSETRUNSTATE.Handle      := TaskInfoDO.Handle;

    ToBusInterface.NewInst(pPara:=#tempCmd, pResult:=#_result);

    if _result.aData[0]$t_BusIFRetvalErrorcode <> _BUS_IF_RETVAL_OK then
      // remember the log message and write it in cyclic priority to avoid a rt runtime error
      CyclicMsgMarker.PostIt.TaskInfoRunFailed := TRUE;
    end_if;
  end_if;
#endif

  // set runstate of read
  dataSETRUNSTATE.Handle      := ISOReadDO.Handle;

  ToBusInterface.NewInst(pPara:=#tempCmd, pResult:=#_result);

  if _result.aData[0]$t_BusIFRetvalErrorcode <> _BUS_IF_RETVAL_OK then
    // remember the log message and write it in cyclic priority to avoid a rt runtime error
    CyclicMsgMarker.PostIt.IsoReadRunFailed := TRUE;
  end_if;

  // set runstate of write
  dataSETRUNSTATE.Handle      := ISOWriteDO.Handle;

  ToBusInterface.NewInst(pPara:=#tempCmd, pResult:=#_result);

  if _result.aData[0]$t_BusIFRetvalErrorcode <> _BUS_IF_RETVAL_OK then
    // remember the log message and write it in cyclic priority to avoid a rt runtime error
    CyclicMsgMarker.PostIt.IsoWriteRunFailed := TRUE;
  end_if;

END_FUNCTION

FUNCTION VIRTUAL GLOBAL SdiasManager::BusIFLogIn
  VAR
  	tempCmd         : CmdStruct;
    _result         : results;
    dataADDCallback : t_BusIFAddCallback;
  END_VAR

  // first check if the module may be deactivated
  tempCmd.uiCmd     := _BUS_IF_GET_DEACTIVATED_STATE;
  ToBusInterface.NewInst(pPara:=#tempCmd, pResult:=#_result);
  if _result.aData[0]$t_BusIFRetvalErrorcode = _BUS_IF_RETVAL_OK then
    b_Deactivated := _result.aData[4]$BOOL;
    if b_Deactivated then
#ifdef HWC_LogError
      HWC_LogError(this, "@00D5 (SdiasManager::BusIFLogIn) SDIAS Manager object inactive");
#endif
      return;
    end_if;
  else
#ifdef HWC_LogError
    HWC_LogError(this, "@00D6 (SdiasManager::BusIFLogIn) Failed to get deactivation state via BusInterface");
#endif
  end_if;

  // Set this class as the operator class of the BusInterface
  dataADDCallback.pthis := this$pVirtualBase;

  tempCmd.uiCmd     := _BUS_IF_ADD_CALLBACK;
  tempCmd.aPara[0]  := (#dataADDCallback)$DINT;
  ToBusInterface.NewInst(pPara:=#tempCmd, pResult:=#_result);
  if _result.aData[0]$t_BusIFRetvalErrorcode <> _BUS_IF_RETVAL_OK then
#ifdef HWC_LogError
    HWC_LogError(this, "@00D7 (SdiasManager::BusIFLogIn) Failed to install callback at bus interface");
#endif
  else
    b_CallbackAdded := TRUE;
  end_if;

END_FUNCTION

FUNCTION VIRTUAL SdiasManager::SendPostInitFinished
	VAR_INPUT
		DisableThisObject 	: BOOL;(* := FALSE *)
	END_VAR
  VAR
  	tempCmd         : CmdStruct;
    _result         : results;
  END_VAR

  b_PostInitFinished := TRUE;
  tempCmd.uiCmd := _BUS_IF_POST_INIT_FINISHED;
  ToBusInterface.NewInst(pPara:=#tempCmd, pResult:=#_result);

  if _result.aData[0]$t_BusIFRetvalErrorcode <> _BUS_IF_RETVAL_OK then
#ifdef HWC_LogError
    HWC_LogError(this, "@00D8 (SdiasManager::CyWork) Failed to set the post init to finished via bus interface!");
#endif
  end_if;

  if DisableThisObject then
    // tell the manager that we don't need to be called for rt syncing
    tempCmd.uiCmd := _BUS_IF_RT_SYNC_READY;
    ToBusInterface.NewInst(pPara:=#tempCmd, pResult:=#_result);

    if _result.aData[0]$t_BusIFRetvalErrorcode <> _BUS_IF_RETVAL_OK then
#ifdef HWC_LogError
      HWC_LogError(this, "@00D9 (SdiasManager::CyWork) Failed to set rt sync ready via bus interface!");
#endif
    end_if;
  end_if;

END_FUNCTION

FUNCTION VIRTUAL SdiasManager::FarMemoryAccessAvailable
	VAR_OUTPUT
		IsAvailable 	: BOOL;
	END_VAR

  if FarMemoryAccessInfo.IsAvailableIsValid = FALSE then
    // get it when entering the first time
    FarMemoryAccessInfo.IsAvailable := FeatureInfo.OptionBits.FarMemoryAccessSupported;
    if (ConnectionType = SDIAS_CON_LOCAL_uC) & (pSDIAS^.udVersion < SDIAS_CIL_VERSION_SUPPORTS_DYNAMIC_DO) then
      // far memory access needs the new CIL
      FarMemoryAccessInfo.IsAvailable := FALSE;
    end_if;
    FarMemoryAccessInfo.IsAvailableIsValid := TRUE;
    if FarMemoryAccessInfo.IsAvailable = FALSE then
#ifdef HWC_LogError
      HWC_LogError(this, "@00DB (SdiasManager::FarMemoryAccessAvailable) Failed to add far memory access! Update OS and/or fpga.");
#endif
    end_if;
  end_if;

  IsAvailable := FarMemoryAccessInfo.IsAvailable;

END_FUNCTION

FUNCTION VIRTUAL SdiasManager::SendTimeBroadCast
  VAR
  	tempCmd             : CmdStruct;
    _result             : results;
    uiBroadCastTime     : UINT;
  END_VAR

  if SupportedFeatures.TimeBroadCastSupported then
    // Get Timestamp from HWControl
    tempCmd.uiCmd := CMD_GET_HW_TIMESTAMP;
    tempCmd.aPara[0]$t_GetHwTimestampCmd.udVersion    := 1;
    tempCmd.aPara[0]$t_GetHwTimestampCmd.udCoreSelect := 0;

    ToBusInterface.NewInst(#tempCmd, #_result);

    // Update Timestamp, do not inkrement here because application accesses this variable!
    uiHWTimestamp := _result.aData[0]$t_GetHwTimestampResult.uiTimeStamp;

    uiBroadCastTime := (uiHWTimestamp + uiSDIASSyncoffset_us) AND 16#7FFF;

    // Inkrement and Boadcast Timestamp
    if aBroadCastTime[0].pWriteData then
      aBroadCastTime[0].pWriteData^ := uiBroadCastTime;
    end_if;
    if aBroadCastTime[1].pWriteData then
      aBroadCastTime[1].pWriteData^ := uiBroadCastTime;
    end_if;
  end_if;

END_FUNCTION

FUNCTION VIRTUAL SdiasManager::SendSyncCntDown
	VAR_OUTPUT
		SyncCountDown 	: UINT;
	END_VAR

  if SupportedFeatures.TimeBroadCastSupported then

    // Decrement before sending, return value is the sent value
    uiSyncCountDown -= 1;

    // Send Sync countdown
    if aBroadCastTime[0].pWriteData then
      aBroadCastTime[0].pWriteData^ := uiSyncCountDown;
    end_if;
    if aBroadCastTime[1].pWriteData then
      aBroadCastTime[1].pWriteData^ := uiSyncCountDown;
    end_if;

  end_if;

  SyncCountDown := uiSyncCountDown;

END_FUNCTION
